LIN {X 0,Y 378.118,Z 312.233,A -85,B 0,C 180,E1 -14679.383,E2 -14679.383} C_VEL
LIN {X 0,Y 374.987,Z 310.362,A -85,B 0,C 180,E1 -14680.649,E2 -14680.649} C_VEL
LIN {X 0,Y 371.579,Z 307.37,A -85,B 0,C 180,E1 -14681.941,E2 -14681.941} C_VEL
LIN {X 0,Y 368.941,Z 304.589,A -85,B 0,C 180,E1 -14682.864,E2 -14682.864} C_VEL
LIN {X 0,Y 365.212,Z 301.597,A -85,B 0,C 180,E1 -14683.991,E2 -14683.991} C_VEL
LIN {X 0,Y 361.301,Z 297.475,A -85,B 0,C 180,E1 -14685.117,E2 -14685.117} C_VEL
LIN {X 0,Y 357.11,Z 293.614,A -85,B 0,C 180,E1 -14686.197,E2 -14686.197} C_VEL
LIN {X 0,Y 354.383,Z 290.674,A -85,B 0,C 180,E1 -14686.85,E2 -14686.85} C_VEL
LIN {X 0,Y 350.827,Z 287.024,A -85,B 0,C 180,E1 -14687.67,E2 -14687.67} C_VEL
LIN {X 0,Y 348.359,Z 284.254,A -85,B 0,C 180,E1 -14688.225,E2 -14688.225} C_VEL
LIN {X 0,Y 345.121,Z 280.43,A -85,B 0,C 180,E1 -14688.925,E2 -14688.925} C_VEL
LIN {X 0,Y 340.974,Z 275.499,A -85,B 0,C 180,E1 -14689.77,E2 -14689.77} C_VEL
LIN {X 0,Y 339.656,Z 273.734,A -85,B 0,C 180,E1 -14690.037,E2 -14690.037} C_VEL
LIN {X 0,Y 337.259,Z 270.621,A -85,B 0,C 180,E1 -14690.505,E2 -14690.505} C_VEL
LIN {X 0,Y 336.338,Z 269.13,A -85,B 0,C 180,E1 -14690.687,E2 -14690.687} C_VEL
LIN {X 0,Y 334.367,Z 266.713,A -85,B 0,C 180,E1 -14691.057,E2 -14691.057} C_VEL
LIN {X 0,Y 333.668,Z 264.421,A -85,B 0,C 180,E1 -14691.262,E2 -14691.262} C_VEL
LIN {X 0,Y 333.674,Z 264.419,A -85,B 0,C 180,E1 -14695.108,E2 -14695.108} C_VEL
LIN {X 0,Y 333.658,Z 264.421,A -85,B 0,C 180,E1 -14698.976,E2 -14698.976} C_VEL
LIN {X 0,Y 333.6,Z 264.429,A -85,B 0,C 180,E1 -14702.594,E2 -14702.594} C_VEL
LIN {X 0,Y 333.627,Z 264.428,A -85,B 0,C 180,E1 -14706.144,E2 -14706.144} C_VEL
LIN {X 0,Y 333.635,Z 264.424,A -85,B 0,C 180,E1 -14709.193,E2 -14709.193} C_VEL
LIN {X 0,Y 333.658,Z 264.42,A -85,B 0,C 180,E1 -14712.519,E2 -14712.519} C_VEL
LIN {X 0,Y 333.687,Z 264.419,A -85,B 0,C 180,E1 -14715.983,E2 -14715.983} C_VEL
LIN {X 0,Y 333.662,Z 264.423,A -85,B 0,C 180,E1 -14719.311,E2 -14719.311} C_VEL
LIN {X 0,Y 333.628,Z 264.427,A -85,B 0,C 180,E1 -14723.175,E2 -14723.175} C_VEL
LIN {X 0,Y 333.639,Z 264.428,A -85,B 0,C 180,E1 -14725.348,E2 -14725.348} C_VEL
LIN {X 0,Y 333.66,Z 264.422,A -85,B 0,C 180,E1 -14729.644,E2 -14729.644} C_VEL
LIN {X 0,Y 333.711,Z 264.414,A -85,B 0,C 180,E1 -14732.408,E2 -14732.408} C_VEL
LIN {X 0,Y 333.7,Z 264.419,A -85,B 0,C 180,E1 -14735.098,E2 -14735.098} C_VEL
LIN {X 0,Y 333.65,Z 264.425,A -85,B 0,C 180,E1 -14739.026,E2 -14739.026} C_VEL
LIN {X 0,Y 333.642,Z 264.421,A -85,B 0,C 180,E1 -14739.892,E2 -14739.892} C_VEL
LIN {X 0,Y 333.012,Z 264.505,A -85,B 0,C 180,E1 -14740.899,E2 -14740.899} C_VEL
LIN {X 0,Y 330.2,Z 264.856,A -85,B 0,C 180,E1 -14742.539,E2 -14742.539} C_VEL
LIN {X 0,Y 327.813,Z 265.154,A -85,B 0,C 180,E1 -14743.868,E2 -14743.868} C_VEL
LIN {X 0,Y 326.808,Z 265.277,A -85,B 0,C 180,E1 -14744.896,E2 -14744.896} C_VEL
LIN {X 0,Y 326.737,Z 265.283,A -85,B 0,C 180,E1 -14745.244,E2 -14745.244} C_VEL
LIN {X 0,Y 326.743,Z 265.284,A -85,B 0,C 180,E1 -14748.846,E2 -14748.846} C_VEL
LIN {X 0,Y 326.928,Z 265.264,A -85,B 0,C 180,E1 -14752.597,E2 -14752.597} C_VEL
LIN {X 0,Y 326.751,Z 265.28,A -85,B 0,C 180,E1 -14755.072,E2 -14755.072} C_VEL
LIN {X 0,Y 327.009,Z 265.244,A -85,B 0,C 180,E1 -14757.544,E2 -14757.544} C_VEL
LIN {X 0,Y 327.039,Z 265.244,A -85,B 0,C 180,E1 -14761.238,E2 -14761.238} C_VEL
LIN {X 0,Y 326.744,Z 265.283,A -85,B 0,C 180,E1 -14763.707,E2 -14763.707} C_VEL
LIN {X 0,Y 326.937,Z 265.263,A -85,B 0,C 180,E1 -14766.177,E2 -14766.177} C_VEL
LIN {X 0,Y 326.783,Z 265.281,A -85,B 0,C 180,E1 -14769.914,E2 -14769.914} C_VEL
LIN {X 0,Y 326.745,Z 265.285,A -85,B 0,C 180,E1 -14773.692,E2 -14773.692} C_VEL
LIN {X 0,Y 326.635,Z 265.299,A -85,B 0,C 180,E1 -14777.538,E2 -14777.538} C_VEL
LIN {X 0,Y 326.614,Z 265.301,A -85,B 0,C 180,E1 -14781.463,E2 -14781.463} C_VEL
LIN {X 0,Y 326.607,Z 265.304,A -85,B 0,C 180,E1 -14785.497,E2 -14785.497} C_VEL
LIN {X 0,Y 326.598,Z 265.301,A -85,B 0,C 180,E1 -14788.262,E2 -14788.262} C_VEL
LIN {X 0,Y 326.582,Z 265.306,A -85,B 0,C 180,E1 -14791.102,E2 -14791.102} C_VEL
LIN {X 0,Y 326.617,Z 265.301,A -85,B 0,C 180,E1 -14794.025,E2 -14794.025} C_VEL
LIN {X 0,Y 326.696,Z 265.699,A -85,B 0,C 180,E1 -14795.515,E2 -14795.515} C_VEL
LIN {X 0,Y 327.042,Z 268.418,A -85,B 0,C 180,E1 -14799.321,E2 -14799.321} C_VEL
LIN {X 0,Y 327.515,Z 271.566,A -85,B 0,C 180,E1 -14803.374,E2 -14803.374} C_VEL
LIN {X 0,Y 327.812,Z 274.541,A -85,B 0,C 180,E1 -14806.803,E2 -14806.803} C_VEL
LIN {X 0,Y 327.68,Z 277.535,A -85,B 0,C 180,E1 -14809.953,E2 -14809.953} C_VEL
LIN {X 0,Y 327.245,Z 280.671,A -85,B 0,C 180,E1 -14813.035,E2 -14813.035} C_VEL
LIN {X 0,Y 326.824,Z 283.847,A -85,B 0,C 180,E1 -14816.007,E2 -14816.007} C_VEL
LIN {X 0,Y 326.327,Z 287.744,A -85,B 0,C 180,E1 -14819.49,E2 -14819.49} C_VEL
LIN {X 0,Y 325.872,Z 291.916,A -85,B 0,C 180,E1 -14823.071,E2 -14823.071} C_VEL
LIN {X 0,Y 325.594,Z 295.184,A -85,B 0,C 180,E1 -14825.788,E2 -14825.788} C_VEL
LIN {X 0,Y 325.375,Z 297.414,A -85,B 0,C 180,E1 -14827.655,E2 -14827.655} C_VEL
LIN {X 0,Y 327.631,Z 306.627,A -85,B 0,C 180,E1 -14828.169,E2 -14828.169} C_VEL
LIN {X 0,Y 329.542,Z 316.235,A -85,B 0,C 180,E1 -14828.811,E2 -14828.811} C_VEL
LIN {X 0,Y 331.065,Z 325.863,A -85,B 0,C 180,E1 -14829.575,E2 -14829.575} C_VEL
LIN {X 0,Y 332.055,Z 334.461,A -85,B 0,C 180,E1 -14830.367,E2 -14830.367} C_VEL
LIN {X 0,Y 332.381,Z 339.384,A -85,B 0,C 180,E1 -14830.869,E2 -14830.869} C_VEL
LIN {X 0,Y 330.863,Z 351.576,A -85,B 0,C 180,E1 -14832.221,E2 -14832.221} C_VEL
LIN {X 0,Y 329.881,Z 359.328,A -85,B 0,C 180,E1 -14833.286,E2 -14833.286} C_VEL
LIN {X 0,Y 328.683,Z 368.467,A -85,B 0,C 180,E1 -14834.815,E2 -14834.815} C_VEL
LIN {X 0,Y 327.874,Z 374.673,A -85,B 0,C 180,E1 -14836.046,E2 -14836.046} C_VEL
LIN {X 0,Y 326.889,Z 381.211,A -85,B 0,C 180,E1 -14837.585,E2 -14837.585} C_VEL
LIN {X 0,Y 326.349,Z 385.716,A -85,B 0,C 180,E1 -14838.825,E2 -14838.825} C_VEL
LIN {X 0,Y 325.657,Z 391.211,A -85,B 0,C 180,E1 -14840.685,E2 -14840.685} C_VEL
LIN {X 0,Y 325.219,Z 395.539,A -85,B 0,C 180,E1 -14842.55,E2 -14842.55} C_VEL
LIN {X 0,Y 325.008,Z 398.409,A -85,B 0,C 180,E1 -14844.139,E2 -14844.139} C_VEL
LIN {X 0,Y 324.915,Z 401.1,A -85,B 0,C 180,E1 -14846.279,E2 -14846.279} C_VEL
LIN {X 0,Y 324.845,Z 402.158,A -85,B 0,C 180,E1 -14847.52,E2 -14847.52} C_VEL
LIN {X 0,Y 324.823,Z 402.747,A -85,B 0,C 180,E1 -14848.76,E2 -14848.76} C_VEL
LIN {X 0,Y 324.823,Z 402.747,A -85,B 0,C 180,E1 -14851.24,E2 -14851.24} C_VEL
LIN {X 0,Y 324.845,Z 402.158,A -85,B 0,C 180,E1 -14852.48,E2 -14852.48} C_VEL
LIN {X 0,Y 324.926,Z 399.709,A -85,B 0,C 180,E1 -14854.963,E2 -14854.963} C_VEL
LIN {X 0,Y 325.108,Z 396.757,A -85,B 0,C 180,E1 -14856.828,E2 -14856.828} C_VEL
LIN {X 0,Y 325.489,Z 392.766,A -85,B 0,C 180,E1 -14858.693,E2 -14858.693} C_VEL
LIN {X 0,Y 326.087,Z 387.633,A -85,B 0,C 180,E1 -14860.556,E2 -14860.556} C_VEL
LIN {X 0,Y 326.724,Z 382.367,A -85,B 0,C 180,E1 -14862.106,E2 -14862.106} C_VEL
LIN {X 0,Y 327.65,Z 376.049,A -85,B 0,C 180,E1 -14863.647,E2 -14863.647} C_VEL
LIN {X 0,Y 328.433,Z 370.094,A -85,B 0,C 180,E1 -14864.879,E2 -14864.879} C_VEL
LIN {X 0,Y 329.506,Z 362.015,A -85,B 0,C 180,E1 -14866.288,E2 -14866.288} C_VEL
LIN {X 0,Y 330.538,Z 353.845,A -85,B 0,C 180,E1 -14867.477,E2 -14867.477} C_VEL
LIN {X 0,Y 331.678,Z 345.117,A -85,B 0,C 180,E1 -14868.532,E2 -14868.532} C_VEL
LIN {X 0,Y 332.396,Z 337.747,A -85,B 0,C 180,E1 -14869.291,E2 -14869.291} C_VEL
LIN {X 0,Y 331.343,Z 327.774,A -85,B 0,C 180,E1 -14870.254,E2 -14870.254} C_VEL
LIN {X 0,Y 330.031,Z 319.039,A -85,B 0,C 180,E1 -14870.98,E2 -14870.98} C_VEL
LIN {X 0,Y 328.032,Z 308.528,A -85,B 0,C 180,E1 -14871.714,E2 -14871.714} C_VEL
LIN {X 0,Y 325.669,Z 299.128,A -85,B 0,C 180,E1 -14872.271,E2 -14872.271} C_VEL
LIN {X 0,Y 325.394,Z 297.387,A -85,B 0,C 180,E1 -14872.368,E2 -14872.368} C_VEL
LIN {X 0,Y 325.704,Z 293.555,A -85,B 0,C 180,E1 -14875.566,E2 -14875.566} C_VEL
LIN {X 0,Y 326.073,Z 290.285,A -85,B 0,C 180,E1 -14878.305,E2 -14878.305} C_VEL
LIN {X 0,Y 326.618,Z 285.433,A -85,B 0,C 180,E1 -14882.543,E2 -14882.543} C_VEL
LIN {X 0,Y 327.059,Z 282.248,A -85,B 0,C 180,E1 -14885.463,E2 -14885.463} C_VEL
LIN {X 0,Y 327.465,Z 279.094,A -85,B 0,C 180,E1 -14888.49,E2 -14888.49} C_VEL
LIN {X 0,Y 327.82,Z 275.972,A -85,B 0,C 180,E1 -14891.65,E2 -14891.65} C_VEL
LIN {X 0,Y 327.845,Z 274.426,A -85,B 0,C 180,E1 -14893.312,E2 -14893.312} C_VEL
LIN {X 0,Y 327.486,Z 271.384,A -85,B 0,C 180,E1 -14896.856,E2 -14896.856} C_VEL
LIN {X 0,Y 327.041,Z 268.391,A -85,B 0,C 180,E1 -14900.679,E2 -14900.679} C_VEL
LIN {X 0,Y 326.666,Z 265.471,A -85,B 0,C 180,E1 -14904.838,E2 -14904.838} C_VEL
LIN {X 0,Y 326.616,Z 265.3,A -85,B 0,C 180,E1 -14907.45,E2 -14907.45} C_VEL
LIN {X 0,Y 326.589,Z 265.305,A -85,B 0,C 180,E1 -14910.328,E2 -14910.328} C_VEL
LIN {X 0,Y 326.603,Z 265.301,A -85,B 0,C 180,E1 -14913.129,E2 -14913.129} C_VEL
LIN {X 0,Y 326.597,Z 265.301,A -85,B 0,C 180,E1 -14917.205,E2 -14917.205} C_VEL
LIN {X 0,Y 326.653,Z 265.293,A -85,B 0,C 180,E1 -14921.2,E2 -14921.2} C_VEL
LIN {X 0,Y 326.728,Z 265.284,A -85,B 0,C 180,E1 -14925.453,E2 -14925.453} C_VEL
LIN {X 0,Y 326.758,Z 265.28,A -85,B 0,C 180,E1 -14928.832,E2 -14928.832} C_VEL
LIN {X 0,Y 326.91,Z 265.261,A -85,B 0,C 180,E1 -14932.582,E2 -14932.582} C_VEL
LIN {X 0,Y 326.741,Z 265.282,A -85,B 0,C 180,E1 -14935.057,E2 -14935.057} C_VEL
LIN {X 0,Y 327.003,Z 265.253,A -85,B 0,C 180,E1 -14937.529,E2 -14937.529} C_VEL
LIN {X 0,Y 327.021,Z 265.245,A -85,B 0,C 180,E1 -14941.224,E2 -14941.224} C_VEL
LIN {X 0,Y 326.758,Z 265.282,A -85,B 0,C 180,E1 -14943.692,E2 -14943.692} C_VEL
LIN {X 0,Y 326.923,Z 265.259,A -85,B 0,C 180,E1 -14946.578,E2 -14946.578} C_VEL
LIN {X 0,Y 326.769,Z 265.279,A -85,B 0,C 180,E1 -14949.9,E2 -14949.9} C_VEL
LIN {X 0,Y 326.74,Z 265.283,A -85,B 0,C 180,E1 -14953.678,E2 -14953.678} C_VEL
LIN {X 0,Y 326.644,Z 265.296,A -85,B 0,C 180,E1 -14957.522,E2 -14957.522} C_VEL
LIN {X 0,Y 326.611,Z 265.297,A -85,B 0,C 180,E1 -14960.129,E2 -14960.129} C_VEL
LIN {X 0,Y 326.623,Z 265.296,A -85,B 0,C 180,E1 -14964.122,E2 -14964.122} C_VEL
LIN {X 0,Y 326.655,Z 265.297,A -85,B 0,C 180,E1 -14966.85,E2 -14966.85} C_VEL
LIN {X 0,Y 326.603,Z 265.303,A -85,B 0,C 180,E1 -14970.602,E2 -14970.602} C_VEL
LIN {X 0,Y 326.573,Z 265.303,A -85,B 0,C 180,E1 -14974.012,E2 -14974.012} C_VEL
LIN {X 0,Y 326.59,Z 265.301,A -85,B 0,C 180,E1 -14977.231,E2 -14977.231} C_VEL
LIN {X 0,Y 326.596,Z 265.303,A -85,B 0,C 180,E1 -14980.196,E2 -14980.196} C_VEL
LIN {X 0,Y 326.616,Z 265.298,A -85,B 0,C 180,E1 -14983.503,E2 -14983.503} C_VEL
LIN {X 0,Y 326.606,Z 265.299,A -85,B 0,C 180,E1 -14987.008,E2 -14987.008} C_VEL
LIN {X 0,Y 326.596,Z 265.301,A -85,B 0,C 180,E1 -14990.76,E2 -14990.76} C_VEL
LIN {X 0,Y 326.563,Z 265.306,A -85,B 0,C 180,E1 -14994.475,E2 -14994.475} C_VEL
LIN {X 0,Y 326.564,Z 265.306,A -85,B 0,C 180,E1 -14997.451,E2 -14997.451} C_VEL
LIN {X 0,Y 326.609,Z 265.301,A -85,B 0,C 180,E1 -15000.336,E2 -15000.336} C_VEL
LIN {X 0,Y 326.639,Z 265.296,A -85,B 0,C 180,E1 -15004.513,E2 -15004.513} C_VEL
LIN {X 0,Y 326.659,Z 265.306,A -85,B 0,C 180,E1 -15007.838,E2 -15007.838} C_VEL
LIN {X 0,Y 327.653,Z 268.102,A -85,B 0,C 180,E1 -15008.036,E2 -15008.036} C_VEL
LIN {X 0,Y 329.492,Z 270.637,A -85,B 0,C 180,E1 -15008.359,E2 -15008.359} C_VEL
LIN {X 0,Y 331.912,Z 274.086,A -85,B 0,C 180,E1 -15008.791,E2 -15008.791} C_VEL
LIN {X 0,Y 336.088,Z 279.409,A -85,B 0,C 180,E1 -15009.56,E2 -15009.56} C_VEL
LIN {X 0,Y 340.074,Z 284.308,A -85,B 0,C 180,E1 -15010.336,E2 -15010.336} C_VEL
LIN {X 0,Y 345.247,Z 290.242,A -85,B 0,C 180,E1 -15011.402,E2 -15011.402} C_VEL
LIN {X 0,Y 350.921,Z 296.303,A -85,B 0,C 180,E1 -15012.674,E2 -15012.674} C_VEL
LIN {X 0,Y 353.867,Z 299.363,A -85,B 0,C 180,E1 -15013.385,E2 -15013.385} C_VEL
LIN {X 0,Y 358.117,Z 303.441,A -85,B 0,C 180,E1 -15014.474,E2 -15014.474} C_VEL
LIN {X 0,Y 360.414,Z 305.696,A -85,B 0,C 180,E1 -15015.099,E2 -15015.099} C_VEL
LIN {X 0,Y 364.679,Z 309.798,A -85,B 0,C 180,E1 -15016.367,E2 -15016.367} C_VEL
LIN {X 0,Y 367.684,Z 312.27,A -85,B 0,C 180,E1 -15017.333,E2 -15017.333} C_VEL
LIN {X 0,Y 370.703,Z 315.447,A -85,B 0,C 180,E1 -15018.461,E2 -15018.461} C_VEL
LIN {X 0,Y 372.499,Z 316.817,A -85,B 0,C 180,E1 -15019.125,E2 -15019.125} C_VEL
LIN {X 0,Y 375.47,Z 318.694,A -85,B 0,C 180,E1 -15020.302,E2 -15020.302} C_VEL
LIN {X 0,Y 378.606,Z 322.035,A -85,B 0,C 180,E1 -15021.956,E2 -15021.956} C_VEL
LIN {X 0,Y 381.325,Z 324.417,A -85,B 0,C 180,E1 -15023.651,E2 -15023.651} C_VEL
LIN {X 0,Y 382.838,Z 325.369,A -85,B 0,C 180,E1 -15024.734,E2 -15024.734} C_VEL
LIN {X 0,Y 384.098,Z 325.94,A -85,B 0,C 180,E1 -15025.803,E2 -15025.803} C_VEL
LIN {X 0,Y 385.138,Z 326.178,A -85,B 0,C 180,E1 -15026.862,E2 -15026.862} C_VEL
LIN {X 0,Y 385.873,Z 326.376,A -85,B 0,C 180,E1 -15027.912,E2 -15027.912} C_VEL
LIN {X 0,Y 386.479,Z 326.455,A -85,B 0,C 180,E1 -15029.734,E2 -15029.734} C_VEL
LIN {X 0,Y 386.344,Z 326.417,A -85,B 0,C 180,E1 -15031.042,E2 -15031.042} C_VEL
LIN {X 0,Y 385.873,Z 326.359,A -85,B 0,C 180,E1 -15032.088,E2 -15032.088} C_VEL
LIN {X 0,Y 385.147,Z 326.153,A -85,B 0,C 180,E1 -15033.138,E2 -15033.138} C_VEL
LIN {X 0,Y 384.113,Z 325.938,A -85,B 0,C 180,E1 -15034.197,E2 -15034.197} C_VEL
LIN {X 0,Y 381.631,Z 324.642,A -85,B 0,C 180,E1 -15036.132,E2 -15036.132} C_VEL
LIN {X 0,Y 379.595,Z 323.032,A -85,B 0,C 180,E1 -15037.446,E2 -15037.446} C_VEL
LIN {X 0,Y 377,Z 320.236,A -85,B 0,C 180,E1 -15038.94,E2 -15038.94} C_VEL
LIN {X 0,Y 375.398,Z 318.661,A -85,B 0,C 180,E1 -15039.7,E2 -15039.7} C_VEL
LIN {X 0,Y 372.189,Z 316.659,A -85,B 0,C 180,E1 -15040.966,E2 -15040.966} C_VEL
LIN {X 0,Y 368.327,Z 313.092,A -85,B 0,C 180,E1 -15042.418,E2 -15042.418} C_VEL
LIN {X 0,Y 366.165,Z 310.906,A -85,B 0,C 180,E1 -15043.166,E2 -15043.166} C_VEL
LIN {X 0,Y 362.128,Z 307.55,A -85,B 0,C 180,E1 -15044.384,E2 -15044.384} C_VEL
LIN {X 0,Y 358.612,Z 303.811,A -85,B 0,C 180,E1 -15045.398,E2 -15045.398} C_VEL
LIN {X 0,Y 354.435,Z 300.023,A -85,B 0,C 180,E1 -15046.464,E2 -15046.464} C_VEL
LIN {X 0,Y 351.099,Z 296.469,A -85,B 0,C 180,E1 -15047.283,E2 -15047.283} C_VEL
LIN {X 0,Y 347.136,Z 292.244,A -85,B 0,C 180,E1 -15048.194,E2 -15048.194} C_VEL
LIN {X 0,Y 341.992,Z 286.589,A -85,B 0,C 180,E1 -15049.275,E2 -15049.275} C_VEL
LIN {X 0,Y 337.043,Z 280.652,A -85,B 0,C 180,E1 -15050.256,E2 -15050.256} C_VEL
LIN {X 0,Y 333.214,Z 275.765,A -85,B 0,C 180,E1 -15050.979,E2 -15050.979} C_VEL
LIN {X 0,Y 329.744,Z 271.114,A -85,B 0,C 180,E1 -15051.591,E2 -15051.591} C_VEL
LIN {X 0,Y 328.709,Z 269.48,A -85,B 0,C 180,E1 -15051.782,E2 -15051.782} C_VEL
LIN {X 0,Y 327.076,Z 266.985,A -85,B 0,C 180,E1 -15052.066,E2 -15052.066} C_VEL
LIN {X 0,Y 326.659,Z 265.297,A -85,B 0,C 180,E1 -15052.193,E2 -15052.193} C_VEL
LIN {X 0,Y 326.639,Z 265.296,A -85,B 0,C 180,E1 -15055.487,E2 -15055.487} C_VEL
LIN {X 0,Y 326.609,Z 265.301,A -85,B 0,C 180,E1 -15059.664,E2 -15059.664} C_VEL
LIN {X 0,Y 326.572,Z 265.303,A -85,B 0,C 180,E1 -15062.952,E2 -15062.952} C_VEL
LIN {X 0,Y 326.582,Z 265.302,A -85,B 0,C 180,E1 -15067.052,E2 -15067.052} C_VEL
LIN {X 0,Y 326.589,Z 265.303,A -85,B 0,C 180,E1 -15070.208,E2 -15070.208} C_VEL
LIN {X 0,Y 326.614,Z 265.301,A -85,B 0,C 180,E1 -15073.516,E2 -15073.516} C_VEL
LIN {X 0,Y 326.609,Z 265.299,A -85,B 0,C 180,E1 -15077.021,E2 -15077.021} C_VEL
LIN {X 0,Y 326.604,Z 265.3,A -85,B 0,C 180,E1 -15080.773,E2 -15080.773} C_VEL
LIN {X 0,Y 326.576,Z 265.302,A -85,B 0,C 180,E1 -15084.487,E2 -15084.487} C_VEL
LIN {X 0,Y 326.575,Z 265.306,A -85,B 0,C 180,E1 -15087.463,E2 -15087.463} C_VEL
LIN {X 0,Y 326.618,Z 265.297,A -85,B 0,C 180,E1 -15090.347,E2 -15090.347} C_VEL
LIN {X 0,Y 326.664,Z 265.292,A -85,B 0,C 180,E1 -15094.524,E2 -15094.524} C_VEL
LIN {X 0,Y 326.596,Z 265.302,A -85,B 0,C 180,E1 -15098.551,E2 -15098.551} C_VEL
LIN {X 0,Y 326.687,Z 265.291,A -85,B 0,C 180,E1 -15101.183,E2 -15101.183} C_VEL
LIN {X 0,Y 326.737,Z 265.283,A -85,B 0,C 180,E1 -15105.244,E2 -15105.244} C_VEL
LIN {X 0,Y 326.09,Z 265.366,A -85,B 0,C 180,E1 -15106.273,E2 -15106.273} C_VEL
LIN {X 0,Y 323.219,Z 265.721,A -85,B 0,C 180,E1 -15107.947,E2 -15107.947} C_VEL
LIN {X 0,Y 320.804,Z 266.021,A -85,B 0,C 180,E1 -15109.304,E2 -15109.304} C_VEL
LIN {X 0,Y 319.814,Z 266.147,A -85,B 0,C 180,E1 -15110.355,E2 -15110.355} C_VEL
LIN {X 0,Y 319.76,Z 266.149,A -85,B 0,C 180,E1 -15110.711,E2 -15110.711} C_VEL
LIN {X 0,Y 319.904,Z 266.134,A -85,B 0,C 180,E1 -15113.701,E2 -15113.701} C_VEL
LIN {X 0,Y 319.955,Z 266.121,A -85,B 0,C 180,E1 -15117.49,E2 -15117.49} C_VEL
LIN {X 0,Y 320.007,Z 266.12,A -85,B 0,C 180,E1 -15121.266,E2 -15121.266} C_VEL
LIN {X 0,Y 319.711,Z 266.158,A -85,B 0,C 180,E1 -15125.052,E2 -15125.052} C_VEL
LIN {X 0,Y 319.85,Z 266.142,A -85,B 0,C 180,E1 -15127.583,E2 -15127.583} C_VEL
LIN {X 0,Y 319.714,Z 266.159,A -85,B 0,C 180,E1 -15131.417,E2 -15131.417} C_VEL
LIN {X 0,Y 319.667,Z 266.164,A -85,B 0,C 180,E1 -15134.684,E2 -15134.684} C_VEL
LIN {X 0,Y 319.591,Z 266.177,A -85,B 0,C 180,E1 -15137.937,E2 -15137.937} C_VEL
LIN {X 0,Y 319.569,Z 266.179,A -85,B 0,C 180,E1 -15141.961,E2 -15141.961} C_VEL
LIN {X 0,Y 319.557,Z 266.179,A -85,B 0,C 180,E1 -15146.101,E2 -15146.101} C_VEL
LIN {X 0,Y 319.533,Z 266.183,A -85,B 0,C 180,E1 -15148.946,E2 -15148.946} C_VEL
LIN {X 0,Y 319.533,Z 266.185,A -85,B 0,C 180,E1 -15151.868,E2 -15151.868} C_VEL
LIN {X 0,Y 319.639,Z 266.435,A -85,B 0,C 180,E1 -15154.873,E2 -15154.873} C_VEL
LIN {X 0,Y 319.891,Z 268.555,A -85,B 0,C 180,E1 -15157.97,E2 -15157.97} C_VEL
LIN {X 0,Y 320.3,Z 271.316,A -85,B 0,C 180,E1 -15161.754,E2 -15161.754} C_VEL
LIN {X 0,Y 320.673,Z 274.349,A -85,B 0,C 180,E1 -15165.468,E2 -15165.468} C_VEL
LIN {X 0,Y 320.773,Z 276.743,A -85,B 0,C 180,E1 -15168.16,E2 -15168.16} C_VEL
LIN {X 0,Y 320.571,Z 278.992,A -85,B 0,C 180,E1 -15170.523,E2 -15170.523} C_VEL
LIN {X 0,Y 319.987,Z 282.879,A -85,B 0,C 180,E1 -15174.363,E2 -15174.363} C_VEL
LIN {X 0,Y 319.422,Z 286.912,A -85,B 0,C 180,E1 -15178.127,E2 -15178.127} C_VEL
LIN {X 0,Y 318.984,Z 291.03,A -85,B 0,C 180,E1 -15181.808,E2 -15181.808} C_VEL
LIN {X 0,Y 318.557,Z 294.987,A -85,B 0,C 180,E1 -15185.218,E2 -15185.218} C_VEL
LIN {X 0,Y 318.335,Z 297.213,A -85,B 0,C 180,E1 -15187.127,E2 -15187.127} C_VEL
LIN {X 0,Y 320.755,Z 307.18,A -85,B 0,C 180,E1 -15187.714,E2 -15187.714} C_VEL
LIN {X 0,Y 322.582,Z 315.881,A -85,B 0,C 180,E1 -15188.322,E2 -15188.322} C_VEL
LIN {X 0,Y 324.268,Z 326.481,A -85,B 0,C 180,E1 -15189.196,E2 -15189.196} C_VEL
LIN {X 0,Y 325.264,Z 335.884,A -85,B 0,C 180,E1 -15190.105,E2 -15190.105} C_VEL
LIN {X 0,Y 325.512,Z 340.784,A -85,B 0,C 180,E1 -15190.613,E2 -15190.613} C_VEL
LIN {X 0,Y 324.085,Z 351.364,A -85,B 0,C 180,E1 -15191.837,E2 -15191.837} C_VEL
LIN {X 0,Y 323.002,Z 359.496,A -85,B 0,C 180,E1 -15192.984,E2 -15192.984} C_VEL
LIN {X 0,Y 322.054,Z 366.823,A -85,B 0,C 180,E1 -15194.209,E2 -15194.209} C_VEL
LIN {X 0,Y 320.974,Z 374.461,A -85,B 0,C 180,E1 -15195.74,E2 -15195.74} C_VEL
LIN {X 0,Y 319.933,Z 380.999,A -85,B 0,C 180,E1 -15197.311,E2 -15197.311} C_VEL
LIN {X 0,Y 319.33,Z 385.503,A -85,B 0,C 180,E1 -15198.576,E2 -15198.576} C_VEL
LIN {X 0,Y 318.637,Z 390.999,A -85,B 0,C 180,E1 -15200.478,E2 -15200.478} C_VEL
LIN {X 0,Y 318.142,Z 395.327,A -85,B 0,C 180,E1 -15202.383,E2 -15202.383} C_VEL
LIN {X 0,Y 317.896,Z 398.501,A -85,B 0,C 180,E1 -15204.222,E2 -15204.222} C_VEL
LIN {X 0,Y 317.824,Z 400.888,A -85,B 0,C 180,E1 -15206.196,E2 -15206.196} C_VEL
LIN {X 0,Y 317.768,Z 401.947,A -85,B 0,C 180,E1 -15207.465,E2 -15207.465} C_VEL
LIN {X 0,Y 317.736,Z 402.536,A -85,B 0,C 180,E1 -15208.733,E2 -15208.733} C_VEL
LIN {X 0,Y 317.736,Z 402.536,A -85,B 0,C 180,E1 -15211.267,E2 -15211.267} C_VEL
LIN {X 0,Y 317.768,Z 401.947,A -85,B 0,C 180,E1 -15212.535,E2 -15212.535} C_VEL
LIN {X 0,Y 317.844,Z 399.498,A -85,B 0,C 180,E1 -15215.074,E2 -15215.074} C_VEL
LIN {X 0,Y 318.035,Z 396.545,A -85,B 0,C 180,E1 -15216.981,E2 -15216.981} C_VEL
LIN {X 0,Y 318.44,Z 392.554,A -85,B 0,C 180,E1 -15218.887,E2 -15218.887} C_VEL
LIN {X 0,Y 319.072,Z 387.421,A -85,B 0,C 180,E1 -15220.791,E2 -15220.791} C_VEL
LIN {X 0,Y 319.762,Z 382.155,A -85,B 0,C 180,E1 -15222.374,E2 -15222.374} C_VEL
LIN {X 0,Y 320.739,Z 375.837,A -85,B 0,C 180,E1 -15223.947,E2 -15223.947} C_VEL
LIN {X 0,Y 321.548,Z 369.882,A -85,B 0,C 180,E1 -15225.205,E2 -15225.205} C_VEL
LIN {X 0,Y 322.568,Z 362.564,A -85,B 0,C 180,E1 -15226.519,E2 -15226.519} C_VEL
LIN {X 0,Y 323.602,Z 354.768,A -85,B 0,C 180,E1 -15227.701,E2 -15227.701} C_VEL
LIN {X 0,Y 324.749,Z 346.256,A -85,B 0,C 180,E1 -15228.778,E2 -15228.778} C_VEL
LIN {X 0,Y 325.585,Z 339.17,A -85,B 0,C 180,E1 -15229.547,E2 -15229.547} C_VEL
LIN {X 0,Y 324.513,Z 328.622,A -85,B 0,C 180,E1 -15230.613,E2 -15230.613} C_VEL
LIN {X 0,Y 322.95,Z 318.107,A -85,B 0,C 180,E1 -15231.508,E2 -15231.508} C_VEL
LIN {X 0,Y 320.929,Z 307.94,A -85,B 0,C 180,E1 -15232.237,E2 -15232.237} C_VEL
LIN {X 0,Y 318.336,Z 297.213,A -85,B 0,C 180,E1 -15232.873,E2 -15232.873} C_VEL
LIN {X 0,Y 318.672,Z 293.356,A -85,B 0,C 180,E1 -15236.172,E2 -15236.172} C_VEL
LIN {X 0,Y 319.05,Z 290.114,A -85,B 0,C 180,E1 -15238.987,E2 -15238.987} C_VEL
LIN {X 0,Y 319.422,Z 286.9,A -85,B 0,C 180,E1 -15241.873,E2 -15241.873} C_VEL
LIN {X 0,Y 320.014,Z 282.866,A -85,B 0,C 180,E1 -15245.644,E2 -15245.644} C_VEL
LIN {X 0,Y 320.572,Z 278.991,A -85,B 0,C 180,E1 -15249.477,E2 -15249.477} C_VEL
LIN {X 0,Y 320.793,Z 275.883,A -85,B 0,C 180,E1 -15252.777,E2 -15252.777} C_VEL
LIN {X 0,Y 320.513,Z 272.817,A -85,B 0,C 180,E1 -15256.352,E2 -15256.352} C_VEL
LIN {X 0,Y 320.09,Z 269.859,A -85,B 0,C 180,E1 -15260.215,E2 -15260.215} C_VEL
LIN {X 0,Y 319.687,Z 266.875,A -85,B 0,C 180,E1 -15264.429,E2 -15264.429} C_VEL
LIN {X 0,Y 319.639,Z 266.424,A -85,B 0,C 180,E1 -15265.127,E2 -15265.127} C_VEL
LIN {X 0,Y 319.533,Z 266.184,A -85,B 0,C 180,E1 -15268.132,E2 -15268.132} C_VEL
LIN {X 0,Y 319.553,Z 266.179,A -85,B 0,C 180,E1 -15271.608,E2 -15271.608} C_VEL
LIN {X 0,Y 319.532,Z 266.182,A -85,B 0,C 180,E1 -15275.292,E2 -15275.292} C_VEL
LIN {X 0,Y 319.569,Z 266.18,A -85,B 0,C 180,E1 -15278.039,E2 -15278.039} C_VEL
LIN {X 0,Y 319.591,Z 266.177,A -85,B 0,C 180,E1 -15282.063,E2 -15282.063} C_VEL
LIN {X 0,Y 319.712,Z 266.162,A -85,B 0,C 180,E1 -15286,E2 -15286} C_VEL
LIN {X 0,Y 319.735,Z 266.159,A -85,B 0,C 180,E1 -15289.865,E2 -15289.865} C_VEL
LIN {X 0,Y 319.894,Z 266.139,A -85,B 0,C 180,E1 -15293.686,E2 -15293.686} C_VEL
LIN {X 0,Y 319.949,Z 266.131,A -85,B 0,C 180,E1 -15297.475,E2 -15297.475} C_VEL
LIN {X 0,Y 319.991,Z 266.121,A -85,B 0,C 180,E1 -15301.251,E2 -15301.251} C_VEL
LIN {X 0,Y 319.708,Z 266.16,A -85,B 0,C 180,E1 -15303.774,E2 -15303.774} C_VEL
LIN {X 0,Y 319.886,Z 266.135,A -85,B 0,C 180,E1 -15306.566,E2 -15306.566} C_VEL
LIN {X 0,Y 319.721,Z 266.156,A -85,B 0,C 180,E1 -15310.12,E2 -15310.12} C_VEL
LIN {X 0,Y 319.714,Z 266.157,A -85,B 0,C 180,E1 -15313.985,E2 -15313.985} C_VEL
LIN {X 0,Y 319.604,Z 266.171,A -85,B 0,C 180,E1 -15317.921,E2 -15317.921} C_VEL
LIN {X 0,Y 319.545,Z 266.178,A -85,B 0,C 180,E1 -15321.947,E2 -15321.947} C_VEL
LIN {X 0,Y 319.591,Z 266.172,A -85,B 0,C 180,E1 -15326.082,E2 -15326.082} C_VEL
LIN {X 0,Y 319.551,Z 266.182,A -85,B 0,C 180,E1 -15328.927,E2 -15328.927} C_VEL
LIN {X 0,Y 319.498,Z 266.184,A -85,B 0,C 180,E1 -15331.855,E2 -15331.855} C_VEL
LIN {X 0,Y 319.544,Z 266.178,A -85,B 0,C 180,E1 -15335.535,E2 -15335.535} C_VEL
LIN {X 0,Y 319.544,Z 266.18,A -85,B 0,C 180,E1 -15338,E2 -15338} C_VEL
LIN {X 0,Y 319.561,Z 266.177,A -85,B 0,C 180,E1 -15341.605,E2 -15341.605} C_VEL
LIN {X 0,Y 319.603,Z 266.171,A -85,B 0,C 180,E1 -15345.279,E2 -15345.279} C_VEL
LIN {X 0,Y 319.538,Z 266.181,A -85,B 0,C 180,E1 -15348.714,E2 -15348.714} C_VEL
LIN {X 0,Y 319.534,Z 266.184,A -85,B 0,C 180,E1 -15352.338,E2 -15352.338} C_VEL
LIN {X 0,Y 319.51,Z 266.183,A -85,B 0,C 180,E1 -15355.118,E2 -15355.118} C_VEL
LIN {X 0,Y 319.522,Z 266.182,A -85,B 0,C 180,E1 -15359.052,E2 -15359.052} C_VEL
LIN {X 0,Y 319.555,Z 266.179,A -85,B 0,C 180,E1 -15362.494,E2 -15362.494} C_VEL
LIN {X 0,Y 319.574,Z 266.178,A -85,B 0,C 180,E1 -15365.302,E2 -15365.302} C_VEL
LIN {X 0,Y 319.61,Z 266.173,A -85,B 0,C 180,E1 -15367.027,E2 -15367.027} C_VEL
LIN {X 0,Y 320.674,Z 269.144,A -85,B 0,C 180,E1 -15367.226,E2 -15367.226} C_VEL
LIN {X 0,Y 322.157,Z 271.338,A -85,B 0,C 180,E1 -15367.45,E2 -15367.45} C_VEL
LIN {X 0,Y 324.428,Z 274.689,A -85,B 0,C 180,E1 -15367.817,E2 -15367.817} C_VEL
LIN {X 0,Y 327.539,Z 279.052,A -85,B 0,C 180,E1 -15368.327,E2 -15368.327} C_VEL
LIN {X 0,Y 332.288,Z 284.974,A -85,B 0,C 180,E1 -15369.174,E2 -15369.174} C_VEL
LIN {X 0,Y 336.349,Z 289.91,A -85,B 0,C 180,E1 -15369.955,E2 -15369.955} C_VEL
LIN {X 0,Y 341.731,Z 296.056,A -85,B 0,C 180,E1 -15371.059,E2 -15371.059} C_VEL
LIN {X 0,Y 347.373,Z 302.107,A -85,B 0,C 180,E1 -15372.334,E2 -15372.334} C_VEL
LIN {X 0,Y 350.5,Z 305.354,A -85,B 0,C 180,E1 -15373.09,E2 -15373.09} C_VEL
LIN {X 0,Y 355.015,Z 309.675,A -85,B 0,C 180,E1 -15374.252,E2 -15374.252} C_VEL
LIN {X 0,Y 360.386,Z 315.045,A -85,B 0,C 180,E1 -15375.805,E2 -15375.805} C_VEL
LIN {X 0,Y 364.886,Z 318.868,A -85,B 0,C 180,E1 -15377.223,E2 -15377.223} C_VEL
LIN {X 0,Y 367.679,Z 321.741,A -85,B 0,C 180,E1 -15378.273,E2 -15378.273} C_VEL
LIN {X 0,Y 371.402,Z 324.359,A -85,B 0,C 180,E1 -15379.679,E2 -15379.679} C_VEL
LIN {X 0,Y 373.699,Z 326.209,A -85,B 0,C 180,E1 -15380.696,E2 -15380.696} C_VEL
LIN {X 0,Y 376.827,Z 329.568,A -85,B 0,C 180,E1 -15382.499,E2 -15382.499} C_VEL
LIN {X 0,Y 378.571,Z 330.947,A -85,B 0,C 180,E1 -15383.605,E2 -15383.605} C_VEL
LIN {X 0,Y 380.766,Z 332.224,A -85,B 0,C 180,E1 -15385.23,E2 -15385.23} C_VEL
LIN {X 0,Y 382.485,Z 332.74,A -85,B 0,C 180,E1 -15386.84,E2 -15386.84} C_VEL
LIN {X 0,Y 383.244,Z 332.949,A -85,B 0,C 180,E1 -15387.898,E2 -15387.898} C_VEL
LIN {X 0,Y 383.734,Z 333.009,A -85,B 0,C 180,E1 -15388.951,E2 -15388.951} C_VEL
LIN {X 0,Y 383.886,Z 333.049,A -85,B 0,C 180,E1 -15390,E2 -15390} C_VEL
LIN {X 0,Y 383.725,Z 333.003,A -85,B 0,C 180,E1 -15391.049,E2 -15391.049} C_VEL
LIN {X 0,Y 383.235,Z 332.95,A -85,B 0,C 180,E1 -15392.102,E2 -15392.102} C_VEL
LIN {X 0,Y 382.491,Z 332.724,A -85,B 0,C 180,E1 -15393.16,E2 -15393.16} C_VEL
LIN {X 0,Y 380.768,Z 332.205,A -85,B 0,C 180,E1 -15394.774,E2 -15394.774} C_VEL
LIN {X 0,Y 378.558,Z 330.954,A -85,B 0,C 180,E1 -15396.395,E2 -15396.395} C_VEL
LIN {X 0,Y 376.064,Z 328.756,A -85,B 0,C 180,E1 -15397.983,E2 -15397.983} C_VEL
LIN {X 0,Y 372.696,Z 325.246,A -85,B 0,C 180,E1 -15399.771,E2 -15399.771} C_VEL
LIN {X 0,Y 369.713,Z 323.369,A -85,B 0,C 180,E1 -15400.958,E2 -15400.958} C_VEL
LIN {X 0,Y 366.503,Z 320.578,A -85,B 0,C 180,E1 -15402.177,E2 -15402.177} C_VEL
LIN {X 0,Y 361.742,Z 316.162,A -85,B 0,C 180,E1 -15403.775,E2 -15403.775} C_VEL
LIN {X 0,Y 358.439,Z 313.187,A -85,B 0,C 180,E1 -15404.767,E2 -15404.767} C_VEL
LIN {X 0,Y 355.431,Z 310.006,A -85,B 0,C 180,E1 -15405.642,E2 -15405.642} C_VEL
LIN {X 0,Y 350.626,Z 305.484,A -85,B 0,C 180,E1 -15406.88,E2 -15406.88} C_VEL
LIN {X 0,Y 347.035,Z 301.806,A -85,B 0,C 180,E1 -15407.747,E2 -15407.747} C_VEL
LIN {X 0,Y 340.82,Z 295.137,A -85,B 0,C 180,E1 -15409.124,E2 -15409.124} C_VEL
LIN {X 0,Y 333.372,Z 286.437,A -85,B 0,C 180,E1 -15410.619,E2 -15410.619} C_VEL
LIN {X 0,Y 328.823,Z 280.611,A -85,B 0,C 180,E1 -15411.453,E2 -15411.453} C_VEL
LIN {X 0,Y 325.211,Z 275.892,A -85,B 0,C 180,E1 -15412.062,E2 -15412.062} C_VEL
LIN {X 0,Y 322.15,Z 271.367,A -85,B 0,C 180,E1 -15412.55,E2 -15412.55} C_VEL
LIN {X 0,Y 319.945,Z 267.598,A -85,B 0,C 180,E1 -15412.889,E2 -15412.889} C_VEL
LIN {X 0,Y 319.592,Z 266.175,A -85,B 0,C 180,E1 -15412.972,E2 -15412.972} C_VEL
LIN {X 0,Y 319.582,Z 266.179,A -85,B 0,C 180,E1 -15416.092,E2 -15416.092} C_VEL
LIN {X 0,Y 319.537,Z 266.18,A -85,B 0,C 180,E1 -15418.938,E2 -15418.938} C_VEL
LIN {X 0,Y 319.487,Z 266.19,A -85,B 0,C 180,E1 -15421.866,E2 -15421.866} C_VEL
LIN {X 0,Y 319.53,Z 266.183,A -85,B 0,C 180,E1 -15425.548,E2 -15425.548} C_VEL
LIN {X 0,Y 319.535,Z 266.184,A -85,B 0,C 180,E1 -15428.013,E2 -15428.013} C_VEL
LIN {X 0,Y 319.557,Z 266.181,A -85,B 0,C 180,E1 -15431.618,E2 -15431.618} C_VEL
LIN {X 0,Y 319.603,Z 266.173,A -85,B 0,C 180,E1 -15435.291,E2 -15435.291} C_VEL
LIN {X 0,Y 319.543,Z 266.179,A -85,B 0,C 180,E1 -15438.727,E2 -15438.727} C_VEL
LIN {X 0,Y 319.544,Z 266.179,A -85,B 0,C 180,E1 -15442.351,E2 -15442.351} C_VEL
LIN {X 0,Y 319.525,Z 266.184,A -85,B 0,C 180,E1 -15445.13,E2 -15445.13} C_VEL
LIN {X 0,Y 319.535,Z 266.184,A -85,B 0,C 180,E1 -15449.067,E2 -15449.067} C_VEL
LIN {X 0,Y 319.577,Z 266.175,A -85,B 0,C 180,E1 -15452.505,E2 -15452.505} C_VEL
LIN {X 0,Y 319.578,Z 266.177,A -85,B 0,C 180,E1 -15455.311,E2 -15455.311} C_VEL
LIN {X 0,Y 319.565,Z 266.175,A -85,B 0,C 180,E1 -15459.407,E2 -15459.407} C_VEL
LIN {X 0,Y 319.604,Z 266.171,A -85,B 0,C 180,E1 -15462.079,E2 -15462.079} C_VEL
LIN {X 0,Y 319.714,Z 266.157,A -85,B 0,C 180,E1 -15466.015,E2 -15466.015} C_VEL
LIN {X 0,Y 319.721,Z 266.156,A -85,B 0,C 180,E1 -15469.88,E2 -15469.88} C_VEL
LIN {X 0,Y 319.76,Z 266.149,A -85,B 0,C 180,E1 -15470.711,E2 -15470.711} C_VEL
LIN {X 0,Y 319.482,Z 266.187,A -85,B 0,C 180,E1 -15471.414,E2 -15471.414} C_VEL
LIN {X 0,Y 317.51,Z 266.44,A -85,B 0,C 180,E1 -15472.793,E2 -15472.793} C_VEL
LIN {X 0,Y 313.709,Z 266.915,A -85,B 0,C 180,E1 -15474.858,E2 -15474.858} C_VEL
LIN {X 0,Y 312.719,Z 267.031,A -85,B 0,C 180,E1 -15475.933,E2 -15475.933} C_VEL
LIN {X 0,Y 312.68,Z 267.032,A -85,B 0,C 180,E1 -15476.298,E2 -15476.298} C_VEL
LIN {X 0,Y 312.96,Z 266.996,A -85,B 0,C 180,E1 -15478.721,E2 -15478.721} C_VEL
LIN {X 0,Y 312.974,Z 266.996,A -85,B 0,C 180,E1 -15481.294,E2 -15481.294} C_VEL
LIN {X 0,Y 312.836,Z 267.017,A -85,B 0,C 180,E1 -15486.457,E2 -15486.457} C_VEL
LIN {X 0,Y 312.751,Z 267.025,A -85,B 0,C 180,E1 -15489.057,E2 -15489.057} C_VEL
LIN {X 0,Y 312.626,Z 267.041,A -85,B 0,C 180,E1 -15492.998,E2 -15492.998} C_VEL
LIN {X 0,Y 312.574,Z 267.051,A -85,B 0,C 180,E1 -15495.66,E2 -15495.66} C_VEL
LIN {X 0,Y 312.534,Z 267.057,A -85,B 0,C 180,E1 -15499.72,E2 -15499.72} C_VEL
LIN {X 0,Y 312.521,Z 267.054,A -85,B 0,C 180,E1 -15502.78,E2 -15502.78} C_VEL
LIN {X 0,Y 312.49,Z 267.058,A -85,B 0,C 180,E1 -15506.738,E2 -15506.738} C_VEL
LIN {X 0,Y 312.478,Z 267.065,A -85,B 0,C 180,E1 -15509.664,E2 -15509.664} C_VEL
LIN {X 0,Y 312.541,Z 267.055,A -85,B 0,C 180,E1 -15513.696,E2 -15513.696} C_VEL
LIN {X 0,Y 312.707,Z 268.308,A -85,B 0,C 180,E1 -15515.994,E2 -15515.994} C_VEL
LIN {X 0,Y 313.105,Z 271.25,A -85,B 0,C 180,E1 -15520.257,E2 -15520.257} C_VEL
LIN {X 0,Y 313.514,Z 274.156,A -85,B 0,C 180,E1 -15524.028,E2 -15524.028} C_VEL
LIN {X 0,Y 313.746,Z 277.243,A -85,B 0,C 180,E1 -15527.671,E2 -15527.671} C_VEL
LIN {X 0,Y 313.42,Z 280.444,A -85,B 0,C 180,E1 -15531.108,E2 -15531.108} C_VEL
LIN {X 0,Y 312.961,Z 283.587,A -85,B 0,C 180,E1 -15534.278,E2 -15534.278} C_VEL
LIN {X 0,Y 312.452,Z 286.77,A -85,B 0,C 180,E1 -15537.328,E2 -15537.328} C_VEL
LIN {X 0,Y 312.064,Z 289.971,A -85,B 0,C 180,E1 -15540.3,E2 -15540.3} C_VEL
LIN {X 0,Y 311.669,Z 293.193,A -85,B 0,C 180,E1 -15543.193,E2 -15543.193} C_VEL
LIN {X 0,Y 311.325,Z 297.107,A -85,B 0,C 180,E1 -15546.593,E2 -15546.593} C_VEL
LIN {X 0,Y 313.531,Z 306.067,A -85,B 0,C 180,E1 -15547.128,E2 -15547.128} C_VEL
LIN {X 0,Y 315.454,Z 314.721,A -85,B 0,C 180,E1 -15547.745,E2 -15547.745} C_VEL
LIN {X 0,Y 317.095,Z 324.833,A -85,B 0,C 180,E1 -15548.583,E2 -15548.583} C_VEL
LIN {X 0,Y 318.2,Z 334.022,A -85,B 0,C 180,E1 -15549.475,E2 -15549.475} C_VEL
LIN {X 0,Y 318.741,Z 340.57,A -85,B 0,C 180,E1 -15550.184,E2 -15550.184} C_VEL
LIN {X 0,Y 317.318,Z 351.152,A -85,B 0,C 180,E1 -15551.435,E2 -15551.435} C_VEL
LIN {X 0,Y 316.243,Z 358.899,A -85,B 0,C 180,E1 -15552.542,E2 -15552.542} C_VEL
LIN {X 0,Y 315.151,Z 366.979,A -85,B 0,C 180,E1 -15553.929,E2 -15553.929} C_VEL
LIN {X 0,Y 314.065,Z 374.249,A -85,B 0,C 180,E1 -15555.419,E2 -15555.419} C_VEL
LIN {X 0,Y 312.994,Z 380.787,A -85,B 0,C 180,E1 -15557.024,E2 -15557.024} C_VEL
LIN {X 0,Y 312.325,Z 385.291,A -85,B 0,C 180,E1 -15558.316,E2 -15558.316} C_VEL
LIN {X 0,Y 311.598,Z 390.787,A -85,B 0,C 180,E1 -15560.261,E2 -15560.261} C_VEL
LIN {X 0,Y 311.076,Z 395.115,A -85,B 0,C 180,E1 -15562.209,E2 -15562.209} C_VEL
LIN {X 0,Y 310.911,Z 397.485,A -85,B 0,C 180,E1 -15563.511,E2 -15563.511} C_VEL
LIN {X 0,Y 310.764,Z 399.286,A -85,B 0,C 180,E1 -15564.81,E2 -15564.81} C_VEL
LIN {X 0,Y 310.692,Z 401.737,A -85,B 0,C 180,E1 -15567.407,E2 -15567.407} C_VEL
LIN {X 0,Y 310.652,Z 402.326,A -85,B 0,C 180,E1 -15568.704,E2 -15568.704} C_VEL
LIN {X 0,Y 310.652,Z 402.326,A -85,B 0,C 180,E1 -15571.296,E2 -15571.296} C_VEL
LIN {X 0,Y 310.692,Z 401.737,A -85,B 0,C 180,E1 -15572.593,E2 -15572.593} C_VEL
LIN {X 0,Y 310.764,Z 399.286,A -85,B 0,C 180,E1 -15575.19,E2 -15575.19} C_VEL
LIN {X 0,Y 310.963,Z 396.333,A -85,B 0,C 180,E1 -15577.14,E2 -15577.14} C_VEL
LIN {X 0,Y 311.411,Z 392.342,A -85,B 0,C 180,E1 -15579.089,E2 -15579.089} C_VEL
LIN {X 0,Y 312.066,Z 387.208,A -85,B 0,C 180,E1 -15581.036,E2 -15581.036} C_VEL
LIN {X 0,Y 312.782,Z 381.942,A -85,B 0,C 180,E1 -15582.655,E2 -15582.655} C_VEL
LIN {X 0,Y 313.823,Z 375.625,A -85,B 0,C 180,E1 -15584.261,E2 -15584.261} C_VEL
LIN {X 0,Y 314.683,Z 369.67,A -85,B 0,C 180,E1 -15585.545,E2 -15585.545} C_VEL
LIN {X 0,Y 315.692,Z 362.74,A -85,B 0,C 180,E1 -15586.822,E2 -15586.822} C_VEL
LIN {X 0,Y 316.812,Z 354.556,A -85,B 0,C 180,E1 -15588.093,E2 -15588.093} C_VEL
LIN {X 0,Y 318.039,Z 346.045,A -85,B 0,C 180,E1 -15589.19,E2 -15589.19} C_VEL
LIN {X 0,Y 318.762,Z 340.571,A -85,B 0,C 180,E1 -15589.815,E2 -15589.815} C_VEL
LIN {X 0,Y 317.726,Z 329.488,A -85,B 0,C 180,E1 -15590.983,E2 -15590.983} C_VEL
LIN {X 0,Y 316.199,Z 318.817,A -85,B 0,C 180,E1 -15591.929,E2 -15591.929} C_VEL
LIN {X 0,Y 314.078,Z 308.274,A -85,B 0,C 180,E1 -15592.721,E2 -15592.721} C_VEL
LIN {X 0,Y 311.376,Z 297.688,A -85,B 0,C 180,E1 -15593.384,E2 -15593.384} C_VEL
LIN {X 0,Y 311.297,Z 297.009,A -85,B 0,C 180,E1 -15593.429,E2 -15593.429} C_VEL
LIN {X 0,Y 311.667,Z 293.158,A -85,B 0,C 180,E1 -15596.807,E2 -15596.807} C_VEL
LIN {X 0,Y 312.064,Z 289.943,A -85,B 0,C 180,E1 -15599.7,E2 -15599.7} C_VEL
LIN {X 0,Y 312.643,Z 285.655,A -85,B 0,C 180,E1 -15603.715,E2 -15603.715} C_VEL
LIN {X 0,Y 313.173,Z 282.007,A -85,B 0,C 180,E1 -15607.294,E2 -15607.294} C_VEL
LIN {X 0,Y 313.617,Z 278.884,A -85,B 0,C 180,E1 -15610.531,E2 -15610.531} C_VEL
LIN {X 0,Y 313.746,Z 277.238,A -85,B 0,C 180,E1 -15612.329,E2 -15612.329} C_VEL
LIN {X 0,Y 313.529,Z 274.248,A -85,B 0,C 180,E1 -15615.831,E2 -15615.831} C_VEL
LIN {X 0,Y 313.135,Z 271.505,A -85,B 0,C 180,E1 -15619.386,E2 -15619.386} C_VEL
LIN {X 0,Y 312.798,Z 269.235,A -85,B 0,C 180,E1 -15622.646,E2 -15622.646} C_VEL
LIN {X 0,Y 312.55,Z 267.162,A -85,B 0,C 180,E1 -15625.789,E2 -15625.789} C_VEL
LIN {X 0,Y 312.516,Z 267.058,A -85,B 0,C 180,E1 -15628.846,E2 -15628.846} C_VEL
LIN {X 0,Y 312.516,Z 267.056,A -85,B 0,C 180,E1 -15631.812,E2 -15631.812} C_VEL
LIN {X 0,Y 312.524,Z 267.058,A -85,B 0,C 180,E1 -15634.699,E2 -15634.699} C_VEL
LIN {X 0,Y 312.546,Z 267.053,A -85,B 0,C 180,E1 -15637.519,E2 -15637.519} C_VEL
LIN {X 0,Y 312.551,Z 267.051,A -85,B 0,C 180,E1 -15641.644,E2 -15641.644} C_VEL
LIN {X 0,Y 312.654,Z 267.039,A -85,B 0,C 180,E1 -15645.678,E2 -15645.678} C_VEL
LIN {X 0,Y 312.686,Z 267.035,A -85,B 0,C 180,E1 -15649.634,E2 -15649.634} C_VEL
LIN {X 0,Y 312.794,Z 267.022,A -85,B 0,C 180,E1 -15652.245,E2 -15652.245} C_VEL
LIN {X 0,Y 312.682,Z 267.033,A -85,B 0,C 180,E1 -15654.835,E2 -15654.835} C_VEL
LIN {X 0,Y 312.974,Z 266.996,A -85,B 0,C 180,E1 -15658.706,E2 -15658.706} C_VEL
LIN {X 0,Y 312.903,Z 266.998,A -85,B 0,C 180,E1 -15662.567,E2 -15662.567} C_VEL
LIN {X 0,Y 312.839,Z 267.013,A -85,B 0,C 180,E1 -15666.549,E2 -15666.549} C_VEL
LIN {X 0,Y 312.738,Z 267.028,A -85,B 0,C 180,E1 -15669.042,E2 -15669.042} C_VEL
LIN {X 0,Y 312.617,Z 267.044,A -85,B 0,C 180,E1 -15672.983,E2 -15672.983} C_VEL
LIN {X 0,Y 312.604,Z 267.044,A -85,B 0,C 180,E1 -15675.643,E2 -15675.643} C_VEL
LIN {X 0,Y 312.539,Z 267.05,A -85,B 0,C 180,E1 -15679.703,E2 -15679.703} C_VEL
LIN {X 0,Y 312.502,Z 267.059,A -85,B 0,C 180,E1 -15682.772,E2 -15682.772} C_VEL
LIN {X 0,Y 312.57,Z 267.046,A -85,B 0,C 180,E1 -15685.925,E2 -15685.925} C_VEL
LIN {X 0,Y 312.508,Z 267.055,A -85,B 0,C 180,E1 -15689.643,E2 -15689.643} C_VEL
LIN {X 0,Y 312.486,Z 267.057,A -85,B 0,C 180,E1 -15693.681,E2 -15693.681} C_VEL
LIN {X 0,Y 312.503,Z 267.056,A -85,B 0,C 180,E1 -15697.376,E2 -15697.376} C_VEL
LIN {X 0,Y 312.488,Z 267.061,A -85,B 0,C 180,E1 -15700.696,E2 -15700.696} C_VEL
LIN {X 0,Y 312.553,Z 267.053,A -85,B 0,C 180,E1 -15704.178,E2 -15704.178} C_VEL
LIN {X 0,Y 312.512,Z 267.056,A -85,B 0,C 180,E1 -15707.898,E2 -15707.898} C_VEL
LIN {X 0,Y 312.496,Z 267.06,A -85,B 0,C 180,E1 -15711.903,E2 -15711.903} C_VEL
LIN {X 0,Y 312.457,Z 267.065,A -85,B 0,C 180,E1 -15715.785,E2 -15715.785} C_VEL
LIN {X 0,Y 312.476,Z 267.06,A -85,B 0,C 180,E1 -15718.849,E2 -15718.849} C_VEL
LIN {X 0,Y 312.522,Z 267.058,A -85,B 0,C 180,E1 -15721.82,E2 -15721.82} C_VEL
LIN {X 0,Y 312.541,Z 267.052,A -85,B 0,C 180,E1 -15724.708,E2 -15724.708} C_VEL
LIN {X 0,Y 312.541,Z 267.079,A -85,B 0,C 180,E1 -15726.357,E2 -15726.357} C_VEL
LIN {X 0,Y 313.557,Z 269.937,A -85,B 0,C 180,E1 -15726.521,E2 -15726.521} C_VEL
LIN {X 0,Y 318.521,Z 277.986,A -85,B 0,C 180,E1 -15727.227,E2 -15727.227} C_VEL
LIN {X 0,Y 323.286,Z 284.384,A -85,B 0,C 180,E1 -15727.988,E2 -15727.988} C_VEL
LIN {X 0,Y 328.139,Z 290.42,A -85,B 0,C 180,E1 -15728.842,E2 -15728.842} C_VEL
LIN {X 0,Y 332.287,Z 295.432,A -85,B 0,C 180,E1 -15729.633,E2 -15729.633} C_VEL
LIN {X 0,Y 337.934,Z 301.856,A -85,B 0,C 180,E1 -15730.806,E2 -15730.806} C_VEL
LIN {X 0,Y 343.66,Z 307.992,A -85,B 0,C 180,E1 -15732.1,E2 -15732.1} C_VEL
LIN {X 0,Y 347.944,Z 312.526,A -85,B 0,C 180,E1 -15733.163,E2 -15733.163} C_VEL
LIN {X 0,Y 352.56,Z 316.579,A -85,B 0,C 180,E1 -15734.345,E2 -15734.345} C_VEL
LIN {X 0,Y 356.935,Z 321.18,A -85,B 0,C 180,E1 -15735.665,E2 -15735.665} C_VEL
LIN {X 0,Y 361.441,Z 325.019,A -85,B 0,C 180,E1 -15737.099,E2 -15737.099} C_VEL
LIN {X 0,Y 365.541,Z 328.902,A -85,B 0,C 180,E1 -15738.628,E2 -15738.628} C_VEL
LIN {X 0,Y 369.423,Z 331.504,A -85,B 0,C 180,E1 -15740.142,E2 -15740.142} C_VEL
LIN {X 0,Y 371.62,Z 333.862,A -85,B 0,C 180,E1 -15741.298,E2 -15741.298} C_VEL
LIN {X 0,Y 373.516,Z 335.802,A -85,B 0,C 180,E1 -15742.432,E2 -15742.432} C_VEL
LIN {X 0,Y 375.287,Z 337.212,A -85,B 0,C 180,E1 -15743.549,E2 -15743.549} C_VEL
LIN {X 0,Y 376.813,Z 338.179,A -85,B 0,C 180,E1 -15744.649,E2 -15744.649} C_VEL
LIN {X 0,Y 378.13,Z 338.782,A -85,B 0,C 180,E1 -15745.737,E2 -15745.737} C_VEL
LIN {X 0,Y 379.795,Z 339.216,A -85,B 0,C 180,E1 -15747.549,E2 -15747.549} C_VEL
LIN {X 0,Y 380.518,Z 339.33,A -85,B 0,C 180,E1 -15748.942,E2 -15748.942} C_VEL
LIN {X 0,Y 380.677,Z 339.36,A -85,B 0,C 180,E1 -15750,E2 -15750} C_VEL
LIN {X 0,Y 380.513,Z 339.315,A -85,B 0,C 180,E1 -15751.058,E2 -15751.058} C_VEL
LIN {X 0,Y 379.795,Z 339.22,A -85,B 0,C 180,E1 -15752.451,E2 -15752.451} C_VEL
LIN {X 0,Y 378.137,Z 338.794,A -85,B 0,C 180,E1 -15754.263,E2 -15754.263} C_VEL
LIN {X 0,Y 376.831,Z 338.183,A -85,B 0,C 180,E1 -15755.351,E2 -15755.351} C_VEL
LIN {X 0,Y 374.955,Z 336.962,A -85,B 0,C 180,E1 -15756.666,E2 -15756.666} C_VEL
LIN {X 0,Y 373.54,Z 335.81,A -85,B 0,C 180,E1 -15757.568,E2 -15757.568} C_VEL
LIN {X 0,Y 370.359,Z 332.457,A -85,B 0,C 180,E1 -15759.393,E2 -15759.393} C_VEL
LIN {X 0,Y 369.432,Z 331.507,A -85,B 0,C 180,E1 -15759.858,E2 -15759.858} C_VEL
LIN {X 0,Y 365.531,Z 328.914,A -85,B 0,C 180,E1 -15761.364,E2 -15761.364} C_VEL
LIN {X 0,Y 363.094,Z 326.767,A -85,B 0,C 180,E1 -15762.293,E2 -15762.293} C_VEL
LIN {X 0,Y 358.266,Z 322.269,A -85,B 0,C 180,E1 -15763.922,E2 -15763.922} C_VEL
LIN {X 0,Y 354.987,Z 319.318,A -85,B 0,C 180,E1 -15764.914,E2 -15764.914} C_VEL
LIN {X 0,Y 350.973,Z 315.28,A -85,B 0,C 180,E1 -15766.056,E2 -15766.056} C_VEL
LIN {X 0,Y 346.503,Z 310.945,A -85,B 0,C 180,E1 -15767.203,E2 -15767.203} C_VEL
LIN {X 0,Y 340.006,Z 304.183,A -85,B 0,C 180,E1 -15768.733,E2 -15768.733} C_VEL
LIN {X 0,Y 333.75,Z 297.144,A -85,B 0,C 180,E1 -15770.07,E2 -15770.07} C_VEL
LIN {X 0,Y 328.666,Z 291.097,A -85,B 0,C 180,E1 -15771.056,E2 -15771.056} C_VEL
LIN {X 0,Y 324.418,Z 285.794,A -85,B 0,C 180,E1 -15771.821,E2 -15771.821} C_VEL
LIN {X 0,Y 320.397,Z 280.562,A -85,B 0,C 180,E1 -15772.485,E2 -15772.485} C_VEL
LIN {X 0,Y 316.838,Z 275.251,A -85,B 0,C 180,E1 -15773.022,E2 -15773.022} C_VEL
LIN {X 0,Y 314.52,Z 271.434,A -85,B 0,C 180,E1 -15773.355,E2 -15773.355} C_VEL
LIN {X 0,Y 312.76,Z 268.115,A -85,B 0,C 180,E1 -15773.597,E2 -15773.597} C_VEL
LIN {X 0,Y 312.524,Z 267.056,A -85,B 0,C 180,E1 -15773.648,E2 -15773.648} C_VEL
LIN {X 0,Y 312.502,Z 267.058,A -85,B 0,C 180,E1 -15776.73,E2 -15776.73} C_VEL
LIN {X 0,Y 312.494,Z 267.059,A -85,B 0,C 180,E1 -15779.655,E2 -15779.655} C_VEL
LIN {X 0,Y 312.47,Z 267.063,A -85,B 0,C 180,E1 -15783.694,E2 -15783.694} C_VEL
LIN {X 0,Y 312.492,Z 267.059,A -85,B 0,C 180,E1 -15787.389,E2 -15787.389} C_VEL
LIN {X 0,Y 312.483,Z 267.058,A -85,B 0,C 180,E1 -15790.709,E2 -15790.709} C_VEL
LIN {X 0,Y 312.552,Z 267.051,A -85,B 0,C 180,E1 -15794.191,E2 -15794.191} C_VEL
LIN {X 0,Y 312.516,Z 267.057,A -85,B 0,C 180,E1 -15797.911,E2 -15797.911} C_VEL
LIN {X 0,Y 312.506,Z 267.057,A -85,B 0,C 180,E1 -15801.916,E2 -15801.916} C_VEL
LIN {X 0,Y 312.473,Z 267.061,A -85,B 0,C 180,E1 -15805.797,E2 -15805.797} C_VEL
LIN {X 0,Y 312.489,Z 267.06,A -85,B 0,C 180,E1 -15808.861,E2 -15808.861} C_VEL
LIN {X 0,Y 312.541,Z 267.051,A -85,B 0,C 180,E1 -15811.832,E2 -15811.832} C_VEL
LIN {X 0,Y 312.559,Z 267.05,A -85,B 0,C 180,E1 -15814.719,E2 -15814.719} C_VEL
LIN {X 0,Y 312.541,Z 267.052,A -85,B 0,C 180,E1 -15817.535,E2 -15817.535} C_VEL
LIN {X 0,Y 312.562,Z 267.048,A -85,B 0,C 180,E1 -15821.661,E2 -15821.661} C_VEL
LIN {X 0,Y 312.668,Z 267.034,A -85,B 0,C 180,E1 -15825.694,E2 -15825.694} C_VEL
LIN {X 0,Y 312.671,Z 267.033,A -85,B 0,C 180,E1 -15829.649,E2 -15829.649} C_VEL
LIN {X 0,Y 312.817,Z 267.019,A -85,B 0,C 180,E1 -15832.261,E2 -15832.261} C_VEL
LIN {X 0,Y 312.69,Z 267.032,A -85,B 0,C 180,E1 -15834.85,E2 -15834.85} C_VEL
LIN {X 0,Y 312.68,Z 267.032,A -85,B 0,C 180,E1 -15836.298,E2 -15836.298} C_VEL
LIN {X 0,Y 312.153,Z 267.092,A -85,B 0,C 180,E1 -15837.375,E2 -15837.375} C_VEL
LIN {X 0,Y 309.436,Z 267.432,A -85,B 0,C 180,E1 -15839.132,E2 -15839.132} C_VEL
LIN {X 0,Y 307.04,Z 267.738,A -85,B 0,C 180,E1 -15840.556,E2 -15840.556} C_VEL
LIN {X 0,Y 305.974,Z 267.868,A -85,B 0,C 180,E1 -15841.657,E2 -15841.657} C_VEL
LIN {X 0,Y 305.871,Z 267.88,A -85,B 0,C 180,E1 -15842.03,E2 -15842.03} C_VEL
LIN {X 0,Y 305.782,Z 267.895,A -85,B 0,C 180,E1 -15846.606,E2 -15846.606} C_VEL
LIN {X 0,Y 305.695,Z 267.904,A -85,B 0,C 180,E1 -15849.268,E2 -15849.268} C_VEL
LIN {X 0,Y 305.573,Z 267.92,A -85,B 0,C 180,E1 -15853.304,E2 -15853.304} C_VEL
LIN {X 0,Y 305.517,Z 267.93,A -85,B 0,C 180,E1 -15856.031,E2 -15856.031} C_VEL
LIN {X 0,Y 305.482,Z 267.932,A -85,B 0,C 180,E1 -15860.194,E2 -15860.194} C_VEL
LIN {X 0,Y 305.447,Z 267.935,A -85,B 0,C 180,E1 -15864.473,E2 -15864.473} C_VEL
LIN {X 0,Y 305.449,Z 267.939,A -85,B 0,C 180,E1 -15867.405,E2 -15867.405} C_VEL
LIN {X 0,Y 305.427,Z 267.94,A -85,B 0,C 180,E1 -15870.42,E2 -15870.42} C_VEL
LIN {X 0,Y 305.484,Z 267.936,A -85,B 0,C 180,E1 -15873.521,E2 -15873.521} C_VEL
LIN {X 0,Y 305.729,Z 269.889,A -85,B 0,C 180,E1 -15876.711,E2 -15876.711} C_VEL
LIN {X 0,Y 306.134,Z 272.686,A -85,B 0,C 180,E1 -15880.749,E2 -15880.749} C_VEL
LIN {X 0,Y 306.523,Z 275.71,A -85,B 0,C 180,E1 -15884.703,E2 -15884.703} C_VEL
LIN {X 0,Y 306.684,Z 277.755,A -85,B 0,C 180,E1 -15887.172,E2 -15887.172} C_VEL
LIN {X 0,Y 306.479,Z 280.329,A -85,B 0,C 180,E1 -15890.054,E2 -15890.054} C_VEL
LIN {X 0,Y 305.968,Z 283.632,A -85,B 0,C 180,E1 -15893.516,E2 -15893.516} C_VEL
LIN {X 0,Y 305.534,Z 286.612,A -85,B 0,C 180,E1 -15896.493,E2 -15896.493} C_VEL
LIN {X 0,Y 305.066,Z 289.798,A -85,B 0,C 180,E1 -15899.548,E2 -15899.548} C_VEL
LIN {X 0,Y 304.674,Z 293.025,A -85,B 0,C 180,E1 -15902.527,E2 -15902.527} C_VEL
LIN {X 0,Y 304.283,Z 296.822,A -85,B 0,C 180,E1 -15906.006,E2 -15906.006} C_VEL
LIN {X 0,Y 306.726,Z 306.799,A -85,B 0,C 180,E1 -15906.639,E2 -15906.639} C_VEL
LIN {X 0,Y 308.868,Z 316.436,A -85,B 0,C 180,E1 -15907.376,E2 -15907.376} C_VEL
LIN {X 0,Y 310.345,Z 325.964,A -85,B 0,C 180,E1 -15908.21,E2 -15908.21} C_VEL
LIN {X 0,Y 311.434,Z 335.445,A -85,B 0,C 180,E1 -15909.181,E2 -15909.181} C_VEL
LIN {X 0,Y 311.897,Z 341.778,A -85,B 0,C 180,E1 -15909.902,E2 -15909.902} C_VEL
LIN {X 0,Y 310.393,Z 352.074,A -85,B 0,C 180,E1 -15911.177,E2 -15911.177} C_VEL
LIN {X 0,Y 309.136,Z 360.607,A -85,B 0,C 180,E1 -15912.469,E2 -15912.469} C_VEL
LIN {X 0,Y 308.056,Z 368.267,A -85,B 0,C 180,E1 -15913.863,E2 -15913.863} C_VEL
LIN {X 0,Y 306.916,Z 375.412,A -85,B 0,C 180,E1 -15915.411,E2 -15915.411} C_VEL
LIN {X 0,Y 305.84,Z 381.73,A -85,B 0,C 180,E1 -15917.053,E2 -15917.053} C_VEL
LIN {X 0,Y 305.072,Z 386.996,A -85,B 0,C 180,E1 -15918.708,E2 -15918.708} C_VEL
LIN {X 0,Y 304.361,Z 392.129,A -85,B 0,C 180,E1 -15920.698,E2 -15920.698} C_VEL
LIN {X 0,Y 303.886,Z 396.121,A -85,B 0,C 180,E1 -15922.692,E2 -15922.692} C_VEL
LIN {X 0,Y 303.687,Z 399.075,A -85,B 0,C 180,E1 -15924.689,E2 -15924.689} C_VEL
LIN {X 0,Y 303.618,Z 401.526,A -85,B 0,C 180,E1 -15927.347,E2 -15927.347} C_VEL
LIN {X 0,Y 303.57,Z 402.115,A -85,B 0,C 180,E1 -15928.673,E2 -15928.673} C_VEL
LIN {X 0,Y 303.57,Z 402.115,A -85,B 0,C 180,E1 -15931.327,E2 -15931.327} C_VEL
LIN {X 0,Y 303.618,Z 401.526,A -85,B 0,C 180,E1 -15932.653,E2 -15932.653} C_VEL
LIN {X 0,Y 303.687,Z 399.075,A -85,B 0,C 180,E1 -15935.311,E2 -15935.311} C_VEL
LIN {X 0,Y 303.886,Z 396.121,A -85,B 0,C 180,E1 -15937.308,E2 -15937.308} C_VEL
LIN {X 0,Y 304.361,Z 392.129,A -85,B 0,C 180,E1 -15939.302,E2 -15939.302} C_VEL
LIN {X 0,Y 305.071,Z 386.996,A -85,B 0,C 180,E1 -15941.292,E2 -15941.292} C_VEL
LIN {X 0,Y 305.832,Z 381.73,A -85,B 0,C 180,E1 -15942.947,E2 -15942.947} C_VEL
LIN {X 0,Y 306.904,Z 375.412,A -85,B 0,C 180,E1 -15944.589,E2 -15944.589} C_VEL
LIN {X 0,Y 308.053,Z 368.279,A -85,B 0,C 180,E1 -15946.135,E2 -15946.135} C_VEL
LIN {X 0,Y 309.148,Z 360.607,A -85,B 0,C 180,E1 -15947.53,E2 -15947.53} C_VEL
LIN {X 0,Y 310.381,Z 352.074,A -85,B 0,C 180,E1 -15948.824,E2 -15948.824} C_VEL
LIN {X 0,Y 311.907,Z 341.778,A -85,B 0,C 180,E1 -15950.097,E2 -15950.097} C_VEL
LIN {X 0,Y 310.906,Z 330.256,A -85,B 0,C 180,E1 -15951.381,E2 -15951.381} C_VEL
LIN {X 0,Y 309.358,Z 319.065,A -85,B 0,C 180,E1 -15952.408,E2 -15952.408} C_VEL
LIN {X 0,Y 307.168,Z 308.457,A -85,B 0,C 180,E1 -15953.241,E2 -15953.241} C_VEL
LIN {X 0,Y 304.334,Z 297.496,A -85,B 0,C 180,E1 -15953.957,E2 -15953.957} C_VEL
LIN {X 0,Y 304.265,Z 296.812,A -85,B 0,C 180,E1 -15954.005,E2 -15954.005} C_VEL
LIN {X 0,Y 304.671,Z 292.978,A -85,B 0,C 180,E1 -15957.474,E2 -15957.474} C_VEL
LIN {X 0,Y 305.245,Z 288.608,A -85,B 0,C 180,E1 -15961.573,E2 -15961.573} C_VEL
LIN {X 0,Y 305.788,Z 285.022,A -85,B 0,C 180,E1 -15965.07,E2 -15965.07} C_VEL
LIN {X 0,Y 306.337,Z 281.46,A -85,B 0,C 180,E1 -15968.729,E2 -15968.729} C_VEL
LIN {X 0,Y 306.651,Z 278.775,A -85,B 0,C 180,E1 -15971.654,E2 -15971.654} C_VEL
LIN {X 0,Y 306.582,Z 276.172,A -85,B 0,C 180,E1 -15974.706,E2 -15974.706} C_VEL
LIN {X 0,Y 306.236,Z 273.392,A -85,B 0,C 180,E1 -15978.269,E2 -15978.269} C_VEL
LIN {X 0,Y 305.873,Z 270.981,A -85,B 0,C 180,E1 -15981.65,E2 -15981.65} C_VEL
LIN {X 0,Y 305.605,Z 268.87,A -85,B 0,C 180,E1 -15984.899,E2 -15984.899} C_VEL
LIN {X 0,Y 305.484,Z 267.936,A -85,B 0,C 180,E1 -15986.479,E2 -15986.479} C_VEL
LIN {X 0,Y 305.427,Z 267.939,A -85,B 0,C 180,E1 -15989.58,E2 -15989.58} C_VEL
LIN {X 0,Y 305.449,Z 267.94,A -85,B 0,C 180,E1 -15992.595,E2 -15992.595} C_VEL
LIN {X 0,Y 305.447,Z 267.937,A -85,B 0,C 180,E1 -15995.527,E2 -15995.527} C_VEL
LIN {X 0,Y 305.482,Z 267.934,A -85,B 0,C 180,E1 -15999.806,E2 -15999.806} C_VEL
LIN {X 0,Y 305.517,Z 267.93,A -85,B 0,C 180,E1 -16003.969,E2 -16003.969} C_VEL
LIN {X 0,Y 305.573,Z 267.92,A -85,B 0,C 180,E1 -16006.696,E2 -16006.696} C_VEL
LIN {X 0,Y 305.753,Z 267.897,A -85,B 0,C 180,E1 -16011.255,E2 -16011.255} C_VEL
LIN {X 0,Y 305.782,Z 267.894,A -85,B 0,C 180,E1 -16013.394,E2 -16013.394} C_VEL
LIN {X 0,Y 305.941,Z 267.872,A -85,B 0,C 180,E1 -16018.676,E2 -16018.676} C_VEL
LIN {X 0,Y 305.929,Z 267.871,A -85,B 0,C 180,E1 -16021.309,E2 -16021.309} C_VEL
LIN {X 0,Y 305.66,Z 267.908,A -85,B 0,C 180,E1 -16025.269,E2 -16025.269} C_VEL
LIN {X 0,Y 305.758,Z 267.897,A -85,B 0,C 180,E1 -16027.919,E2 -16027.919} C_VEL
LIN {X 0,Y 305.582,Z 267.919,A -85,B 0,C 180,E1 -16031.937,E2 -16031.937} C_VEL
LIN {X 0,Y 305.591,Z 267.919,A -85,B 0,C 180,E1 -16035.006,E2 -16035.006} C_VEL
LIN {X 0,Y 305.522,Z 267.925,A -85,B 0,C 180,E1 -16039.418,E2 -16039.418} C_VEL
LIN {X 0,Y 305.463,Z 267.937,A -85,B 0,C 180,E1 -16043.031,E2 -16043.031} C_VEL
LIN {X 0,Y 305.499,Z 267.928,A -85,B 0,C 180,E1 -16046.21,E2 -16046.21} C_VEL
LIN {X 0,Y 305.459,Z 267.937,A -85,B 0,C 180,E1 -16049.039,E2 -16049.039} C_VEL
LIN {X 0,Y 305.41,Z 267.939,A -85,B 0,C 180,E1 -16051.945,E2 -16051.945} C_VEL
LIN {X 0,Y 305.427,Z 267.938,A -85,B 0,C 180,E1 -16055.106,E2 -16055.106} C_VEL
LIN {X 0,Y 305.445,Z 267.939,A -85,B 0,C 180,E1 -16058.529,E2 -16058.529} C_VEL
LIN {X 0,Y 305.481,Z 267.934,A -85,B 0,C 180,E1 -16062.592,E2 -16062.592} C_VEL
LIN {X 0,Y 305.491,Z 267.934,A -85,B 0,C 180,E1 -16066.358,E2 -16066.358} C_VEL
LIN {X 0,Y 305.439,Z 267.938,A -85,B 0,C 180,E1 -16069.89,E2 -16069.89} C_VEL
LIN {X 0,Y 305.436,Z 267.938,A -85,B 0,C 180,E1 -16073.625,E2 -16073.625} C_VEL
LIN {X 0,Y 305.416,Z 267.941,A -85,B 0,C 180,E1 -16076.478,E2 -16076.478} C_VEL
LIN {X 0,Y 305.414,Z 267.942,A -85,B 0,C 180,E1 -16079.586,E2 -16079.586} C_VEL
LIN {X 0,Y 305.469,Z 267.933,A -85,B 0,C 180,E1 -16082.604,E2 -16082.604} C_VEL
LIN {X 0,Y 305.479,Z 267.935,A -85,B 0,C 180,E1 -16085.745,E2 -16085.745} C_VEL
LIN {X 0,Y 306.488,Z 270.763,A -85,B 0,C 180,E1 -16085.919,E2 -16085.919} C_VEL
LIN {X 0,Y 310.96,Z 278.733,A -85,B 0,C 180,E1 -16086.513,E2 -16086.513} C_VEL
LIN {X 0,Y 316.634,Z 287.055,A -85,B 0,C 180,E1 -16087.373,E2 -16087.373} C_VEL
LIN {X 0,Y 323.228,Z 295.22,A -85,B 0,C 180,E1 -16088.494,E2 -16088.494} C_VEL
LIN {X 0,Y 328.123,Z 301.03,A -85,B 0,C 180,E1 -16089.426,E2 -16089.426} C_VEL
LIN {X 0,Y 333.127,Z 306.844,A -85,B 0,C 180,E1 -16090.476,E2 -16090.476} C_VEL
LIN {X 0,Y 339.887,Z 313.966,A -85,B 0,C 180,E1 -16091.986,E2 -16091.986} C_VEL
LIN {X 0,Y 345.677,Z 319.938,A -85,B 0,C 180,E1 -16093.463,E2 -16093.463} C_VEL
LIN {X 0,Y 349.841,Z 323.856,A -85,B 0,C 180,E1 -16094.601,E2 -16094.601} C_VEL
LIN {X 0,Y 352.777,Z 326.843,A -85,B 0,C 180,E1 -16095.492,E2 -16095.492} C_VEL
LIN {X 0,Y 357.384,Z 330.758,A -85,B 0,C 180,E1 -16096.95,E2 -16096.95} C_VEL
LIN {X 0,Y 361.45,Z 334.631,A -85,B 0,C 180,E1 -16098.461,E2 -16098.461} C_VEL
LIN {X 0,Y 365.534,Z 337.433,A -85,B 0,C 180,E1 -16100.036,E2 -16100.036} C_VEL
LIN {X 0,Y 369.023,Z 341.072,A -85,B 0,C 180,E1 -16101.956,E2 -16101.956} C_VEL
LIN {X 0,Y 371.427,Z 343.142,A -85,B 0,C 180,E1 -16103.481,E2 -16103.481} C_VEL
LIN {X 0,Y 373.737,Z 344.522,A -85,B 0,C 180,E1 -16105.189,E2 -16105.189} C_VEL
LIN {X 0,Y 375.441,Z 345.092,A -85,B 0,C 180,E1 -16106.781,E2 -16106.781} C_VEL
LIN {X 0,Y 376.266,Z 345.303,A -85,B 0,C 180,E1 -16107.859,E2 -16107.859} C_VEL
LIN {X 0,Y 376.803,Z 345.371,A -85,B 0,C 180,E1 -16108.931,E2 -16108.931} C_VEL
LIN {X 0,Y 376.97,Z 345.404,A -85,B 0,C 180,E1 -16110,E2 -16110} C_VEL
LIN {X 0,Y 376.794,Z 345.363,A -85,B 0,C 180,E1 -16111.069,E2 -16111.069} C_VEL
LIN {X 0,Y 376.261,Z 345.286,A -85,B 0,C 180,E1 -16112.141,E2 -16112.141} C_VEL
LIN {X 0,Y 375.439,Z 345.073,A -85,B 0,C 180,E1 -16113.219,E2 -16113.219} C_VEL
LIN {X 0,Y 373.735,Z 344.505,A -85,B 0,C 180,E1 -16114.807,E2 -16114.807} C_VEL
LIN {X 0,Y 371.396,Z 343.156,A -85,B 0,C 180,E1 -16116.519,E2 -16116.519} C_VEL
LIN {X 0,Y 369.025,Z 341.072,A -85,B 0,C 180,E1 -16118.046,E2 -16118.046} C_VEL
LIN {X 0,Y 365.533,Z 337.442,A -85,B 0,C 180,E1 -16119.964,E2 -16119.964} C_VEL
LIN {X 0,Y 361.413,Z 334.634,A -85,B 0,C 180,E1 -16121.543,E2 -16121.543} C_VEL
LIN {X 0,Y 357.331,Z 330.755,A -85,B 0,C 180,E1 -16123.059,E2 -16123.059} C_VEL
LIN {X 0,Y 352.729,Z 326.833,A -85,B 0,C 180,E1 -16124.51,E2 -16124.51} C_VEL
LIN {X 0,Y 346.858,Z 320.967,A -85,B 0,C 180,E1 -16126.239,E2 -16126.239} C_VEL
LIN {X 0,Y 341.829,Z 315.956,A -85,B 0,C 180,E1 -16127.536,E2 -16127.536} C_VEL
LIN {X 0,Y 336.703,Z 310.744,A -85,B 0,C 180,E1 -16128.741,E2 -16128.741} C_VEL
LIN {X 0,Y 329.595,Z 302.803,A -85,B 0,C 180,E1 -16130.276,E2 -16130.276} C_VEL
LIN {X 0,Y 323.906,Z 296.058,A -85,B 0,C 180,E1 -16131.375,E2 -16131.375} C_VEL
LIN {X 0,Y 319.531,Z 290.567,A -85,B 0,C 180,E1 -16132.162,E2 -16132.162} C_VEL
LIN {X 0,Y 315.43,Z 285.264,A -85,B 0,C 180,E1 -16132.827,E2 -16132.827} C_VEL
LIN {X 0,Y 310.231,Z 277.606,A -85,B 0,C 180,E1 -16133.587,E2 -16133.587} C_VEL
LIN {X 0,Y 305.888,Z 269.522,A -85,B 0,C 180,E1 -16134.163,E2 -16134.163} C_VEL
LIN {X 0,Y 305.473,Z 267.936,A -85,B 0,C 180,E1 -16134.274,E2 -16134.274} C_VEL
LIN {X 0,Y 305.469,Z 267.933,A -85,B 0,C 180,E1 -16137.396,E2 -16137.396} C_VEL
LIN {X 0,Y 305.414,Z 267.942,A -85,B 0,C 180,E1 -16140.414,E2 -16140.414} C_VEL
LIN {X 0,Y 305.416,Z 267.943,A -85,B 0,C 180,E1 -16144.084,E2 -16144.084} C_VEL
LIN {X 0,Y 305.433,Z 267.937,A -85,B 0,C 180,E1 -16146.744,E2 -16146.744} C_VEL
LIN {X 0,Y 305.441,Z 267.935,A -85,B 0,C 180,E1 -16150.613,E2 -16150.613} C_VEL
LIN {X 0,Y 305.502,Z 267.928,A -85,B 0,C 180,E1 -16154.523,E2 -16154.523} C_VEL
LIN {X 0,Y 305.461,Z 267.934,A -85,B 0,C 180,E1 -16158.16,E2 -16158.16} C_VEL
LIN {X 0,Y 305.471,Z 267.936,A -85,B 0,C 180,E1 -16161.609,E2 -16161.609} C_VEL
LIN {X 0,Y 305.427,Z 267.938,A -85,B 0,C 180,E1 -16164.894,E2 -16164.894} C_VEL
LIN {X 0,Y 305.418,Z 267.938,A -85,B 0,C 180,E1 -16168.364,E2 -16168.364} C_VEL
LIN {X 0,Y 305.484,Z 267.934,A -85,B 0,C 180,E1 -16171.121,E2 -16171.121} C_VEL
LIN {X 0,Y 305.539,Z 267.922,A -85,B 0,C 180,E1 -16174.095,E2 -16174.095} C_VEL
LIN {X 0,Y 305.453,Z 267.935,A -85,B 0,C 180,E1 -16178.409,E2 -16178.409} C_VEL
LIN {X 0,Y 305.523,Z 267.927,A -85,B 0,C 180,E1 -16181.223,E2 -16181.223} C_VEL
LIN {X 0,Y 305.609,Z 267.914,A -85,B 0,C 180,E1 -16185.356,E2 -16185.356} C_VEL
LIN {X 0,Y 305.61,Z 267.913,A -85,B 0,C 180,E1 -16189.407,E2 -16189.407} C_VEL
LIN {X 0,Y 305.758,Z 267.897,A -85,B 0,C 180,E1 -16192.081,E2 -16192.081} C_VEL
LIN {X 0,Y 305.66,Z 267.908,A -85,B 0,C 180,E1 -16194.731,E2 -16194.731} C_VEL
LIN {X 0,Y 305.929,Z 267.871,A -85,B 0,C 180,E1 -16198.691,E2 -16198.691} C_VEL
LIN {X 0,Y 305.871,Z 267.88,A -85,B 0,C 180,E1 -16202.03,E2 -16202.03} C_VEL
LIN {X 0,Y 305.147,Z 267.973,A -85,B 0,C 180,E1 -16203.128,E2 -16203.128} C_VEL
LIN {X 0,Y 302.233,Z 268.336,A -85,B 0,C 180,E1 -16204.913,E2 -16204.913} C_VEL
LIN {X 0,Y 299.797,Z 268.642,A -85,B 0,C 180,E1 -16206.361,E2 -16206.361} C_VEL
LIN {X 0,Y 298.767,Z 268.768,A -85,B 0,C 180,E1 -16207.483,E2 -16207.483} C_VEL
LIN {X 0,Y 298.69,Z 268.779,A -85,B 0,C 180,E1 -16207.863,E2 -16207.863} C_VEL
LIN {X 0,Y 298.546,Z 268.798,A -85,B 0,C 180,E1 -16212.239,E2 -16212.239} C_VEL
LIN {X 0,Y 298.528,Z 268.798,A -85,B 0,C 180,E1 -16215.157,E2 -16215.157} C_VEL
LIN {X 0,Y 298.438,Z 268.812,A -85,B 0,C 180,E1 -16219.618,E2 -16219.618} C_VEL
LIN {X 0,Y 298.39,Z 268.82,A -85,B 0,C 180,E1 -16223.61,E2 -16223.61} C_VEL
LIN {X 0,Y 298.41,Z 268.812,A -85,B 0,C 180,E1 -16226.589,E2 -16226.589} C_VEL
LIN {X 0,Y 298.367,Z 268.823,A -85,B 0,C 180,E1 -16229.654,E2 -16229.654} C_VEL
LIN {X 0,Y 298.408,Z 268.817,A -85,B 0,C 180,E1 -16232.806,E2 -16232.806} C_VEL
LIN {X 0,Y 298.662,Z 270.568,A -85,B 0,C 180,E1 -16236.043,E2 -16236.043} C_VEL
LIN {X 0,Y 298.961,Z 272.788,A -85,B 0,C 180,E1 -16239.406,E2 -16239.406} C_VEL
LIN {X 0,Y 299.36,Z 275.604,A -85,B 0,C 180,E1 -16243.301,E2 -16243.301} C_VEL
LIN {X 0,Y 299.646,Z 278.253,A -85,B 0,C 180,E1 -16246.65,E2 -16246.65} C_VEL
LIN {X 0,Y 299.543,Z 280.212,A -85,B 0,C 180,E1 -16248.934,E2 -16248.934} C_VEL
LIN {X 0,Y 299.087,Z 283.318,A -85,B 0,C 180,E1 -16252.342,E2 -16252.342} C_VEL
LIN {X 0,Y 298.601,Z 286.466,A -85,B 0,C 180,E1 -16255.607,E2 -16255.607} C_VEL
LIN {X 0,Y 298.116,Z 289.638,A -85,B 0,C 180,E1 -16258.759,E2 -16258.759} C_VEL
LIN {X 0,Y 297.682,Z 292.826,A -85,B 0,C 180,E1 -16261.825,E2 -16261.825} C_VEL
LIN {X 0,Y 297.246,Z 296.813,A -85,B 0,C 180,E1 -16265.418,E2 -16265.418} C_VEL
LIN {X 0,Y 299.733,Z 306.576,A -85,B 0,C 180,E1 -16266.061,E2 -16266.061} C_VEL
LIN {X 0,Y 301.969,Z 316.367,A -85,B 0,C 180,E1 -16266.84,E2 -16266.84} C_VEL
LIN {X 0,Y 303.349,Z 324.978,A -85,B 0,C 180,E1 -16267.613,E2 -16267.613} C_VEL
LIN {X 0,Y 304.405,Z 333.582,A -85,B 0,C 180,E1 -16268.499,E2 -16268.499} C_VEL
LIN {X 0,Y 305.034,Z 342.918,A -85,B 0,C 180,E1 -16269.606,E2 -16269.606} C_VEL
LIN {X 0,Y 303.688,Z 351.863,A -85,B 0,C 180,E1 -16270.745,E2 -16270.745} C_VEL
LIN {X 0,Y 302.34,Z 360.394,A -85,B 0,C 180,E1 -16272.062,E2 -16272.062} C_VEL
LIN {X 0,Y 301.315,Z 367.579,A -85,B 0,C 180,E1 -16273.39,E2 -16273.39} C_VEL
LIN {X 0,Y 300.262,Z 373.824,A -85,B 0,C 180,E1 -16274.733,E2 -16274.733} C_VEL
LIN {X 0,Y 299.126,Z 380.363,A -85,B 0,C 180,E1 -16276.412,E2 -16276.412} C_VEL
LIN {X 0,Y 298.345,Z 384.865,A -85,B 0,C 180,E1 -16277.76,E2 -16277.76} C_VEL
LIN {X 0,Y 297.536,Z 390.362,A -85,B 0,C 180,E1 -16279.796,E2 -16279.796} C_VEL
LIN {X 0,Y 296.984,Z 394.691,A -85,B 0,C 180,E1 -16281.837,E2 -16281.837} C_VEL
LIN {X 0,Y 296.757,Z 397.061,A -85,B 0,C 180,E1 -16283.2,E2 -16283.2} C_VEL
LIN {X 0,Y 296.602,Z 398.863,A -85,B 0,C 180,E1 -16284.561,E2 -16284.561} C_VEL
LIN {X 0,Y 296.545,Z 401.315,A -85,B 0,C 180,E1 -16287.283,E2 -16287.283} C_VEL
LIN {X 0,Y 296.491,Z 401.904,A -85,B 0,C 180,E1 -16288.642,E2 -16288.642} C_VEL
LIN {X 0,Y 296.491,Z 401.904,A -85,B 0,C 180,E1 -16291.358,E2 -16291.358} C_VEL
LIN {X 0,Y 296.545,Z 401.315,A -85,B 0,C 180,E1 -16292.717,E2 -16292.717} C_VEL
LIN {X 0,Y 296.622,Z 398.863,A -85,B 0,C 180,E1 -16295.438,E2 -16295.438} C_VEL
LIN {X 0,Y 296.834,Z 395.909,A -85,B 0,C 180,E1 -16297.482,E2 -16297.482} C_VEL
LIN {X 0,Y 297.328,Z 391.917,A -85,B 0,C 180,E1 -16299.524,E2 -16299.524} C_VEL
LIN {X 0,Y 298.059,Z 386.783,A -85,B 0,C 180,E1 -16301.561,E2 -16301.561} C_VEL
LIN {X 0,Y 298.903,Z 381.518,A -85,B 0,C 180,E1 -16303.253,E2 -16303.253} C_VEL
LIN {X 0,Y 300,Z 375.2,A -85,B 0,C 180,E1 -16304.933,E2 -16304.933} C_VEL
LIN {X 0,Y 301.01,Z 369.247,A -85,B 0,C 180,E1 -16306.27,E2 -16306.27} C_VEL
LIN {X 0,Y 302.056,Z 362.315,A -85,B 0,C 180,E1 -16307.606,E2 -16307.606} C_VEL
LIN {X 0,Y 303.319,Z 354.132,A -85,B 0,C 180,E1 -16308.928,E2 -16308.928} C_VEL
LIN {X 0,Y 304.65,Z 345.622,A -85,B 0,C 180,E1 -16310.069,E2 -16310.069} C_VEL
LIN {X 0,Y 305.048,Z 341.561,A -85,B 0,C 180,E1 -16310.569,E2 -16310.569} C_VEL
LIN {X 0,Y 304.074,Z 330.371,A -85,B 0,C 180,E1 -16311.856,E2 -16311.856} C_VEL
LIN {X 0,Y 302.442,Z 318.895,A -85,B 0,C 180,E1 -16312.946,E2 -16312.946} C_VEL
LIN {X 0,Y 300.136,Z 308.081,A -85,B 0,C 180,E1 -16313.827,E2 -16313.827} C_VEL
LIN {X 0,Y 297.32,Z 297.457,A -85,B 0,C 180,E1 -16314.553,E2 -16314.553} C_VEL
LIN {X 0,Y 297.241,Z 296.625,A -85,B 0,C 180,E1 -16314.601,E2 -16314.601} C_VEL
LIN {X 0,Y 297.853,Z 291.759,A -85,B 0,C 180,E1 -16319.177,E2 -16319.177} C_VEL
LIN {X 0,Y 298.347,Z 288.029,A -85,B 0,C 180,E1 -16322.805,E2 -16322.805} C_VEL
LIN {X 0,Y 298.859,Z 284.884,A -85,B 0,C 180,E1 -16326.008,E2 -16326.008} C_VEL
LIN {X 0,Y 299.34,Z 281.757,A -85,B 0,C 180,E1 -16329.339,E2 -16329.339} C_VEL
LIN {X 0,Y 299.67,Z 278.652,A -85,B 0,C 180,E1 -16332.852,E2 -16332.852} C_VEL
LIN {X 0,Y 299.507,Z 276.697,A -85,B 0,C 180,E1 -16335.247,E2 -16335.247} C_VEL
LIN {X 0,Y 299.147,Z 273.989,A -85,B 0,C 180,E1 -16338.859,E2 -16338.859} C_VEL
LIN {X 0,Y 298.789,Z 271.636,A -85,B 0,C 180,E1 -16342.29,E2 -16342.29} C_VEL
LIN {X 0,Y 298.554,Z 269.565,A -85,B 0,C 180,E1 -16345.593,E2 -16345.593} C_VEL
LIN {X 0,Y 298.408,Z 268.818,A -85,B 0,C 180,E1 -16347.194,E2 -16347.194} C_VEL
LIN {X 0,Y 298.374,Z 268.821,A -85,B 0,C 180,E1 -16350.633,E2 -16350.633} C_VEL
LIN {X 0,Y 298.42,Z 268.815,A -85,B 0,C 180,E1 -16354.911,E2 -16354.911} C_VEL
LIN {X 0,Y 298.398,Z 268.817,A -85,B 0,C 180,E1 -16357.855,E2 -16357.855} C_VEL
LIN {X 0,Y 298.458,Z 268.808,A -85,B 0,C 180,E1 -16360.744,E2 -16360.744} C_VEL
LIN {X 0,Y 298.514,Z 268.799,A -85,B 0,C 180,E1 -16364.984,E2 -16364.984} C_VEL
LIN {X 0,Y 298.583,Z 268.79,A -85,B 0,C 180,E1 -16369.139,E2 -16369.139} C_VEL
LIN {X 0,Y 298.697,Z 268.78,A -85,B 0,C 180,E1 -16371.877,E2 -16371.877} C_VEL
LIN {X 0,Y 298.623,Z 268.785,A -85,B 0,C 180,E1 -16374.591,E2 -16374.591} C_VEL
LIN {X 0,Y 298.907,Z 268.748,A -85,B 0,C 180,E1 -16378.645,E2 -16378.645} C_VEL
LIN {X 0,Y 298.897,Z 268.745,A -85,B 0,C 180,E1 -16381.339,E2 -16381.339} C_VEL
LIN {X 0,Y 298.742,Z 268.77,A -85,B 0,C 180,E1 -16386.747,E2 -16386.747} C_VEL
LIN {X 0,Y 298.613,Z 268.788,A -85,B 0,C 180,E1 -16389.474,E2 -16389.474} C_VEL
LIN {X 0,Y 298.528,Z 268.797,A -85,B 0,C 180,E1 -16393.608,E2 -16393.608} C_VEL
LIN {X 0,Y 298.468,Z 268.804,A -85,B 0,C 180,E1 -16396.404,E2 -16396.404} C_VEL
LIN {X 0,Y 298.462,Z 268.803,A -85,B 0,C 180,E1 -16399.631,E2 -16399.631} C_VEL
LIN {X 0,Y 298.405,Z 268.812,A -85,B 0,C 180,E1 -16403.592,E2 -16403.592} C_VEL
LIN {X 0,Y 298.459,Z 268.806,A -85,B 0,C 180,E1 -16406.567,E2 -16406.567} C_VEL
LIN {X 0,Y 298.387,Z 268.814,A -85,B 0,C 180,E1 -16409.634,E2 -16409.634} C_VEL
LIN {X 0,Y 298.363,Z 268.821,A -85,B 0,C 180,E1 -16412.793,E2 -16412.793} C_VEL
LIN {X 0,Y 298.43,Z 268.812,A -85,B 0,C 180,E1 -16416.805,E2 -16416.805} C_VEL
LIN {X 0,Y 298.415,Z 268.811,A -85,B 0,C 180,E1 -16421.243,E2 -16421.243} C_VEL
LIN {X 0,Y 298.447,Z 268.807,A -85,B 0,C 180,E1 -16425.054,E2 -16425.054} C_VEL
LIN {X 0,Y 298.409,Z 268.812,A -85,B 0,C 180,E1 -16428.892,E2 -16428.892} C_VEL
LIN {X 0,Y 298.404,Z 268.812,A -85,B 0,C 180,E1 -16433.185,E2 -16433.185} C_VEL
LIN {X 0,Y 298.348,Z 268.82,A -85,B 0,C 180,E1 -16437.195,E2 -16437.195} C_VEL
LIN {X 0,Y 298.381,Z 268.816,A -85,B 0,C 180,E1 -16440.61,E2 -16440.61} C_VEL
LIN {X 0,Y 298.432,Z 268.812,A -85,B 0,C 180,E1 -16443.47,E2 -16443.47} C_VEL
LIN {X 0,Y 298.434,Z 268.811,A -85,B 0,C 180,E1 -16445.15,E2 -16445.15} C_VEL
LIN {X 0,Y 299.562,Z 271.864,A -85,B 0,C 180,E1 -16445.348,E2 -16445.348} C_VEL
LIN {X 0,Y 304.459,Z 281.322,A -85,B 0,C 180,E1 -16446.05,E2 -16446.05} C_VEL
LIN {X 0,Y 309.593,Z 288.95,A -85,B 0,C 180,E1 -16446.808,E2 -16446.808} C_VEL
LIN {X 0,Y 314.007,Z 294.792,A -85,B 0,C 180,E1 -16447.518,E2 -16447.518} C_VEL
LIN {X 0,Y 320.361,Z 302.867,A -85,B 0,C 180,E1 -16448.666,E2 -16448.666} C_VEL
LIN {X 0,Y 327.104,Z 310.636,A -85,B 0,C 180,E1 -16450.02,E2 -16450.02} C_VEL
LIN {X 0,Y 333.535,Z 317.604,A -85,B 0,C 180,E1 -16451.446,E2 -16451.446} C_VEL
LIN {X 0,Y 340.653,Z 324.898,A -85,B 0,C 180,E1 -16453.212,E2 -16453.212} C_VEL
LIN {X 0,Y 345.037,Z 328.924,A -85,B 0,C 180,E1 -16454.381,E2 -16454.381} C_VEL
LIN {X 0,Y 348.47,Z 332.462,A -85,B 0,C 180,E1 -16455.442,E2 -16455.442} C_VEL
LIN {X 0,Y 353.351,Z 336.715,A -85,B 0,C 180,E1 -16457.011,E2 -16457.011} C_VEL
LIN {X 0,Y 358.157,Z 341.045,A -85,B 0,C 180,E1 -16458.801,E2 -16458.801} C_VEL
LIN {X 0,Y 361.063,Z 342.968,A -85,B 0,C 180,E1 -16459.911,E2 -16459.911} C_VEL
LIN {X 0,Y 363.322,Z 345.262,A -85,B 0,C 180,E1 -16461.098,E2 -16461.098} C_VEL
LIN {X 0,Y 365.248,Z 347.254,A -85,B 0,C 180,E1 -16462.259,E2 -16462.259} C_VEL
LIN {X 0,Y 367.556,Z 349.08,A -85,B 0,C 180,E1 -16463.78,E2 -16463.78} C_VEL
LIN {X 0,Y 369.99,Z 350.409,A -85,B 0,C 180,E1 -16465.643,E2 -16465.643} C_VEL
LIN {X 0,Y 371.172,Z 350.801,A -85,B 0,C 180,E1 -16466.744,E2 -16466.744} C_VEL
LIN {X 0,Y 372.515,Z 351.103,A -85,B 0,C 180,E1 -16468.706,E2 -16468.706} C_VEL
LIN {X 0,Y 372.814,Z 351.138,A -85,B 0,C 180,E1 -16470,E2 -16470} C_VEL
LIN {X 0,Y 372.515,Z 351.089,A -85,B 0,C 180,E1 -16471.297,E2 -16471.297} C_VEL
LIN {X 0,Y 371.176,Z 350.776,A -85,B 0,C 180,E1 -16473.256,E2 -16473.256} C_VEL
LIN {X 0,Y 369.977,Z 350.428,A -85,B 0,C 180,E1 -16474.358,E2 -16474.358} C_VEL
LIN {X 0,Y 367.56,Z 349.09,A -85,B 0,C 180,E1 -16476.225,E2 -16476.225} C_VEL
LIN {X 0,Y 365.258,Z 347.229,A -85,B 0,C 180,E1 -16477.74,E2 -16477.74} C_VEL
LIN {X 0,Y 362.954,Z 344.831,A -85,B 0,C 180,E1 -16479.121,E2 -16479.121} C_VEL
LIN {X 0,Y 361.057,Z 342.963,A -85,B 0,C 180,E1 -16480.089,E2 -16480.089} C_VEL
LIN {X 0,Y 356.25,Z 339.507,A -85,B 0,C 180,E1 -16481.909,E2 -16481.909} C_VEL
LIN {X 0,Y 351.884,Z 335.317,A -85,B 0,C 180,E1 -16483.501,E2 -16483.501} C_VEL
LIN {X 0,Y 347.219,Z 331.274,A -85,B 0,C 180,E1 -16484.947,E2 -16484.947} C_VEL
LIN {X 0,Y 342.08,Z 326.154,A -85,B 0,C 180,E1 -16486.438,E2 -16486.438} C_VEL
LIN {X 0,Y 336.281,Z 320.284,A -85,B 0,C 180,E1 -16487.916,E2 -16487.916} C_VEL
LIN {X 0,Y 330.592,Z 314.311,A -85,B 0,C 180,E1 -16489.244,E2 -16489.244} C_VEL
LIN {X 0,Y 324.731,Z 307.797,A -85,B 0,C 180,E1 -16490.487,E2 -16490.487} C_VEL
LIN {X 0,Y 319.552,Z 301.782,A -85,B 0,C 180,E1 -16491.497,E2 -16491.497} C_VEL
LIN {X 0,Y 312.034,Z 292.438,A -85,B 0,C 180,E1 -16492.801,E2 -16492.801} C_VEL
LIN {X 0,Y 306.443,Z 284.371,A -85,B 0,C 180,E1 -16493.659,E2 -16493.659} C_VEL
LIN {X 0,Y 301.831,Z 276.63,A -85,B 0,C 180,E1 -16494.323,E2 -16494.323} C_VEL
LIN {X 0,Y 298.639,Z 269.773,A -85,B 0,C 180,E1 -16494.789,E2 -16494.789} C_VEL
LIN {X 0,Y 298.443,Z 268.81,A -85,B 0,C 180,E1 -16494.882,E2 -16494.882} C_VEL
LIN {X 0,Y 298.411,Z 268.816,A -85,B 0,C 180,E1 -16498.1,E2 -16498.1} C_VEL
LIN {X 0,Y 298.348,Z 268.824,A -85,B 0,C 180,E1 -16502.023,E2 -16502.023} C_VEL
LIN {X 0,Y 298.373,Z 268.82,A -85,B 0,C 180,E1 -16506.075,E2 -16506.075} C_VEL
LIN {X 0,Y 298.381,Z 268.818,A -85,B 0,C 180,E1 -16509.49,E2 -16509.49} C_VEL
LIN {X 0,Y 298.427,Z 268.81,A -85,B 0,C 180,E1 -16513.124,E2 -16513.124} C_VEL
LIN {X 0,Y 298.43,Z 268.81,A -85,B 0,C 180,E1 -16516.94,E2 -16516.94} C_VEL
LIN {X 0,Y 298.392,Z 268.815,A -85,B 0,C 180,E1 -16521.008,E2 -16521.008} C_VEL
LIN {X 0,Y 298.396,Z 268.814,A -85,B 0,C 180,E1 -16523.939,E2 -16523.939} C_VEL
LIN {X 0,Y 298.362,Z 268.818,A -85,B 0,C 180,E1 -16527.992,E2 -16527.992} C_VEL
LIN {X 0,Y 298.429,Z 268.809,A -85,B 0,C 180,E1 -16531.912,E2 -16531.912} C_VEL
LIN {X 0,Y 298.456,Z 268.807,A -85,B 0,C 180,E1 -16534.932,E2 -16534.932} C_VEL
LIN {X 0,Y 298.408,Z 268.811,A -85,B 0,C 180,E1 -16539.322,E2 -16539.322} C_VEL
LIN {X 0,Y 298.458,Z 268.806,A -85,B 0,C 180,E1 -16542.184,E2 -16542.184} C_VEL
LIN {X 0,Y 298.569,Z 268.793,A -85,B 0,C 180,E1 -16545.003,E2 -16545.003} C_VEL
LIN {X 0,Y 298.569,Z 268.791,A -85,B 0,C 180,E1 -16549.154,E2 -16549.154} C_VEL
LIN {X 0,Y 298.704,Z 268.775,A -85,B 0,C 180,E1 -16551.893,E2 -16551.893} C_VEL
LIN {X 0,Y 298.63,Z 268.785,A -85,B 0,C 180,E1 -16554.607,E2 -16554.607} C_VEL
LIN {X 0,Y 298.897,Z 268.745,A -85,B 0,C 180,E1 -16558.661,E2 -16558.661} C_VEL
LIN {X 0,Y 298.835,Z 268.756,A -85,B 0,C 180,E1 -16562.01,E2 -16562.01} C_VEL
LIN {X 0,Y 298.731,Z 268.772,A -85,B 0,C 180,E1 -16566.763,E2 -16566.763} C_VEL
LIN {X 0,Y 298.69,Z 268.779,A -85,B 0,C 180,E1 -16567.863,E2 -16567.863} C_VEL
LIN {X 0,Y 298.013,Z 268.868,A -85,B 0,C 180,E1 -16568.988,E2 -16568.988} C_VEL
LIN {X 0,Y 295.065,Z 269.231,A -85,B 0,C 180,E1 -16570.815,E2 -16570.815} C_VEL
LIN {X 0,Y 292.578,Z 269.541,A -85,B 0,C 180,E1 -16572.299,E2 -16572.299} C_VEL
LIN {X 0,Y 291.544,Z 269.669,A -85,B 0,C 180,E1 -16573.45,E2 -16573.45} C_VEL
LIN {X 0,Y 291.478,Z 269.678,A -85,B 0,C 180,E1 -16573.84,E2 -16573.84} C_VEL
LIN {X 0,Y 291.409,Z 269.684,A -85,B 0,C 180,E1 -16576.83,E2 -16576.83} C_VEL
LIN {X 0,Y 291.398,Z 269.689,A -85,B 0,C 180,E1 -16579.849,E2 -16579.849} C_VEL
LIN {X 0,Y 291.333,Z 269.694,A -85,B 0,C 180,E1 -16584.218,E2 -16584.218} C_VEL
LIN {X 0,Y 291.338,Z 269.697,A -85,B 0,C 180,E1 -16587.287,E2 -16587.287} C_VEL
LIN {X 0,Y 291.312,Z 269.699,A -85,B 0,C 180,E1 -16590.447,E2 -16590.447} C_VEL
LIN {X 0,Y 291.352,Z 269.697,A -85,B 0,C 180,E1 -16592.408,E2 -16592.408} C_VEL
LIN {X 0,Y 291.608,Z 271.252,A -85,B 0,C 180,E1 -16595.347,E2 -16595.347} C_VEL
LIN {X 0,Y 291.95,Z 274.003,A -85,B 0,C 180,E1 -16599.618,E2 -16599.618} C_VEL
LIN {X 0,Y 292.221,Z 275.903,A -85,B 0,C 180,E1 -16602.338,E2 -16602.338} C_VEL
LIN {X 0,Y 292.572,Z 278.771,A -85,B 0,C 180,E1 -16606.115,E2 -16606.115} C_VEL
LIN {X 0,Y 292.543,Z 280.437,A -85,B 0,C 180,E1 -16608.145,E2 -16608.145} C_VEL
LIN {X 0,Y 292.176,Z 283.181,A -85,B 0,C 180,E1 -16611.289,E2 -16611.289} C_VEL
LIN {X 0,Y 291.627,Z 286.653,A -85,B 0,C 180,E1 -16615.031,E2 -16615.031} C_VEL
LIN {X 0,Y 291.159,Z 289.462,A -85,B 0,C 180,E1 -16617.925,E2 -16617.925} C_VEL
LIN {X 0,Y 290.729,Z 292.639,A -85,B 0,C 180,E1 -16621.088,E2 -16621.088} C_VEL
LIN {X 0,Y 290.24,Z 296.436,A -85,B 0,C 180,E1 -16624.773,E2 -16624.773} C_VEL
LIN {X 0,Y 292.253,Z 304.329,A -85,B 0,C 180,E1 -16625.3,E2 -16625.3} C_VEL
LIN {X 0,Y 294.781,Z 315.05,A -85,B 0,C 180,E1 -16626.162,E2 -16626.162} C_VEL
LIN {X 0,Y 296.318,Z 323.538,A -85,B 0,C 180,E1 -16626.941,E2 -16626.941} C_VEL
LIN {X 0,Y 297.577,Z 333.988,A -85,B 0,C 180,E1 -16628.05,E2 -16628.05} C_VEL
LIN {X 0,Y 298.292,Z 342.717,A -85,B 0,C 180,E1 -16629.126,E2 -16629.126} C_VEL
LIN {X 0,Y 296.982,Z 351.651,A -85,B 0,C 180,E1 -16630.293,E2 -16630.293} C_VEL
LIN {X 0,Y 295.572,Z 360.182,A -85,B 0,C 180,E1 -16631.636,E2 -16631.636} C_VEL
LIN {X 0,Y 294.425,Z 367.717,A -85,B 0,C 180,E1 -16633.066,E2 -16633.066} C_VEL
LIN {X 0,Y 293.366,Z 373.611,A -85,B 0,C 180,E1 -16634.365,E2 -16634.365} C_VEL
LIN {X 0,Y 292.203,Z 380.151,A -85,B 0,C 180,E1 -16636.083,E2 -16636.083} C_VEL
LIN {X 0,Y 291.377,Z 384.653,A -85,B 0,C 180,E1 -16637.463,E2 -16637.463} C_VEL
LIN {X 0,Y 290.527,Z 390.15,A -85,B 0,C 180,E1 -16639.547,E2 -16639.547} C_VEL
LIN {X 0,Y 289.93,Z 394.479,A -85,B 0,C 180,E1 -16641.637,E2 -16641.637} C_VEL
LIN {X 0,Y 289.685,Z 396.849,A -85,B 0,C 180,E1 -16643.033,E2 -16643.033} C_VEL
LIN {X 0,Y 289.519,Z 398.703,A -85,B 0,C 180,E1 -16644.468,E2 -16644.468} C_VEL
LIN {X 0,Y 289.451,Z 401.104,A -85,B 0,C 180,E1 -16647.217,E2 -16647.217} C_VEL
LIN {X 0,Y 289.414,Z 401.693,A -85,B 0,C 180,E1 -16648.609,E2 -16648.609} C_VEL
LIN {X 0,Y 289.414,Z 401.693,A -85,B 0,C 180,E1 -16651.391,E2 -16651.391} C_VEL
LIN {X 0,Y 289.451,Z 401.104,A -85,B 0,C 180,E1 -16652.783,E2 -16652.783} C_VEL
LIN {X 0,Y 289.539,Z 398.652,A -85,B 0,C 180,E1 -16655.572,E2 -16655.572} C_VEL
LIN {X 0,Y 289.767,Z 395.697,A -85,B 0,C 180,E1 -16657.666,E2 -16657.666} C_VEL
LIN {X 0,Y 290.309,Z 391.705,A -85,B 0,C 180,E1 -16659.756,E2 -16659.756} C_VEL
LIN {X 0,Y 291.066,Z 386.571,A -85,B 0,C 180,E1 -16661.843,E2 -16661.843} C_VEL
LIN {X 0,Y 291.978,Z 381.306,A -85,B 0,C 180,E1 -16663.573,E2 -16663.573} C_VEL
LIN {X 0,Y 293.103,Z 374.987,A -85,B 0,C 180,E1 -16665.293,E2 -16665.293} C_VEL
LIN {X 0,Y 294.193,Z 369.035,A -85,B 0,C 180,E1 -16666.658,E2 -16666.658} C_VEL
LIN {X 0,Y 295.268,Z 362.103,A -85,B 0,C 180,E1 -16668.024,E2 -16668.024} C_VEL
LIN {X 0,Y 296.568,Z 353.92,A -85,B 0,C 180,E1 -16669.376,E2 -16669.376} C_VEL
LIN {X 0,Y 297.969,Z 345.41,A -85,B 0,C 180,E1 -16670.539,E2 -16670.539} C_VEL
LIN {X 0,Y 298.165,Z 341.372,A -85,B 0,C 180,E1 -16671.062,E2 -16671.062} C_VEL
LIN {X 0,Y 297.179,Z 330.019,A -85,B 0,C 180,E1 -16672.402,E2 -16672.402} C_VEL
LIN {X 0,Y 295.556,Z 318.831,A -85,B 0,C 180,E1 -16673.501,E2 -16673.501} C_VEL
LIN {X 0,Y 293.157,Z 307.906,A -85,B 0,C 180,E1 -16674.428,E2 -16674.428} C_VEL
LIN {X 0,Y 290.374,Z 297.573,A -85,B 0,C 180,E1 -16675.168,E2 -16675.168} C_VEL
LIN {X 0,Y 290.241,Z 296.437,A -85,B 0,C 180,E1 -16675.226,E2 -16675.226} C_VEL
LIN {X 0,Y 290.804,Z 291.997,A -85,B 0,C 180,E1 -16679.528,E2 -16679.528} C_VEL
LIN {X 0,Y 291.402,Z 287.877,A -85,B 0,C 180,E1 -16683.69,E2 -16683.69} C_VEL
LIN {X 0,Y 291.997,Z 284.366,A -85,B 0,C 180,E1 -16687.405,E2 -16687.405} C_VEL
LIN {X 0,Y 292.389,Z 281.619,A -85,B 0,C 180,E1 -16690.464,E2 -16690.464} C_VEL
LIN {X 0,Y 292.571,Z 280.077,A -85,B 0,C 180,E1 -16692.267,E2 -16692.267} C_VEL
LIN {X 0,Y 292.562,Z 278.533,A -85,B 0,C 180,E1 -16694.157,E2 -16694.157} C_VEL
LIN {X 0,Y 292.223,Z 275.889,A -85,B 0,C 180,E1 -16697.662,E2 -16697.662} C_VEL
LIN {X 0,Y 291.864,Z 273.417,A -85,B 0,C 180,E1 -16701.232,E2 -16701.232} C_VEL
LIN {X 0,Y 291.56,Z 271.026,A -85,B 0,C 180,E1 -16705.04,E2 -16705.04} C_VEL
LIN {X 0,Y 291.377,Z 269.691,A -85,B 0,C 180,E1 -16707.944,E2 -16707.944} C_VEL
LIN {X 0,Y 291.324,Z 269.697,A -85,B 0,C 180,E1 -16711.145,E2 -16711.145} C_VEL
LIN {X 0,Y 291.35,Z 269.697,A -85,B 0,C 180,E1 -16714.258,E2 -16714.258} C_VEL
LIN {X 0,Y 291.357,Z 269.693,A -85,B 0,C 180,E1 -16717.29,E2 -16717.29} C_VEL
LIN {X 0,Y 291.391,Z 269.692,A -85,B 0,C 180,E1 -16720.258,E2 -16720.258} C_VEL
LIN {X 0,Y 291.478,Z 269.676,A -85,B 0,C 180,E1 -16724.676,E2 -16724.676} C_VEL
LIN {X 0,Y 291.529,Z 269.669,A -85,B 0,C 180,E1 -16728.873,E2 -16728.873} C_VEL
LIN {X 0,Y 291.651,Z 269.657,A -85,B 0,C 180,E1 -16731.679,E2 -16731.679} C_VEL
LIN {X 0,Y 291.593,Z 269.661,A -85,B 0,C 180,E1 -16734.46,E2 -16734.46} C_VEL
LIN {X 0,Y 291.873,Z 269.624,A -85,B 0,C 180,E1 -16738.612,E2 -16738.612} C_VEL
LIN {X 0,Y 291.865,Z 269.619,A -85,B 0,C 180,E1 -16741.372,E2 -16741.372} C_VEL
LIN {X 0,Y 291.693,Z 269.649,A -85,B 0,C 180,E1 -16746.911,E2 -16746.911} C_VEL
LIN {X 0,Y 291.555,Z 269.666,A -85,B 0,C 180,E1 -16749.706,E2 -16749.706} C_VEL
LIN {X 0,Y 291.498,Z 269.671,A -85,B 0,C 180,E1 -16753.942,E2 -16753.942} C_VEL
LIN {X 0,Y 291.414,Z 269.684,A -85,B 0,C 180,E1 -16756.813,E2 -16756.813} C_VEL
LIN {X 0,Y 291.403,Z 269.681,A -85,B 0,C 180,E1 -16759.852,E2 -16759.852} C_VEL
LIN {X 0,Y 291.357,Z 269.689,A -85,B 0,C 180,E1 -16764.199,E2 -16764.199} C_VEL
LIN {X 0,Y 291.392,Z 269.688,A -85,B 0,C 180,E1 -16767.264,E2 -16767.264} C_VEL
LIN {X 0,Y 291.304,Z 269.699,A -85,B 0,C 180,E1 -16770.429,E2 -16770.429} C_VEL
LIN {X 0,Y 291.312,Z 269.695,A -85,B 0,C 180,E1 -16773.691,E2 -16773.691} C_VEL
LIN {X 0,Y 291.362,Z 269.69,A -85,B 0,C 180,E1 -16777.252,E2 -16777.252} C_VEL
LIN {X 0,Y 291.363,Z 269.693,A -85,B 0,C 180,E1 -16780.624,E2 -16780.624} C_VEL
LIN {X 0,Y 291.366,Z 269.693,A -85,B 0,C 180,E1 -16784.373,E2 -16784.373} C_VEL
LIN {X 0,Y 291.345,Z 269.695,A -85,B 0,C 180,E1 -16788.384,E2 -16788.384} C_VEL
LIN {X 0,Y 291.332,Z 269.694,A -85,B 0,C 180,E1 -16791.156,E2 -16791.156} C_VEL
LIN {X 0,Y 291.315,Z 269.697,A -85,B 0,C 180,E1 -16794.62,E2 -16794.62} C_VEL
LIN {X 0,Y 291.325,Z 269.699,A -85,B 0,C 180,E1 -16797.946,E2 -16797.946} C_VEL
LIN {X 0,Y 291.331,Z 269.695,A -85,B 0,C 180,E1 -16801.153,E2 -16801.153} C_VEL
LIN {X 0,Y 291.403,Z 269.686,A -85,B 0,C 180,E1 -16804.525,E2 -16804.525} C_VEL
LIN {X 0,Y 292.44,Z 272.615,A -85,B 0,C 180,E1 -16804.72,E2 -16804.72} C_VEL
LIN {X 0,Y 297.903,Z 283.604,A -85,B 0,C 180,E1 -16805.575,E2 -16805.575} C_VEL
LIN {X 0,Y 303.777,Z 292.88,A -85,B 0,C 180,E1 -16806.53,E2 -16806.53} C_VEL
LIN {X 0,Y 311.184,Z 302.758,A -85,B 0,C 180,E1 -16807.787,E2 -16807.787} C_VEL
LIN {X 0,Y 318.195,Z 311.012,A -85,B 0,C 180,E1 -16809.088,E2 -16809.088} C_VEL
LIN {X 0,Y 324.943,Z 318.602,A -85,B 0,C 180,E1 -16810.504,E2 -16810.504} C_VEL
LIN {X 0,Y 330.853,Z 324.914,A -85,B 0,C 180,E1 -16811.883,E2 -16811.883} C_VEL
LIN {X 0,Y 337.13,Z 331.292,A -85,B 0,C 180,E1 -16813.488,E2 -16813.488} C_VEL
LIN {X 0,Y 342.086,Z 336.104,A -85,B 0,C 180,E1 -16814.887,E2 -16814.887} C_VEL
LIN {X 0,Y 348.118,Z 341.499,A -85,B 0,C 180,E1 -16816.812,E2 -16816.812} C_VEL
LIN {X 0,Y 351.797,Z 344.989,A -85,B 0,C 180,E1 -16818.158,E2 -16818.158} C_VEL
LIN {X 0,Y 356.02,Z 348.075,A -85,B 0,C 180,E1 -16819.766,E2 -16819.766} C_VEL
LIN {X 0,Y 359.381,Z 351.355,A -85,B 0,C 180,E1 -16821.547,E2 -16821.547} C_VEL
LIN {X 0,Y 362.154,Z 353.865,A -85,B 0,C 180,E1 -16823.314,E2 -16823.314} C_VEL
LIN {X 0,Y 363.768,Z 354.966,A -85,B 0,C 180,E1 -16824.457,E2 -16824.457} C_VEL
LIN {X 0,Y 366.122,Z 356.052,A -85,B 0,C 180,E1 -16826.384,E2 -16826.384} C_VEL
LIN {X 0,Y 367.396,Z 356.419,A -85,B 0,C 180,E1 -16827.807,E2 -16827.807} C_VEL
LIN {X 0,Y 368.022,Z 356.511,A -85,B 0,C 180,E1 -16828.906,E2 -16828.906} C_VEL
LIN {X 0,Y 368.228,Z 356.538,A -85,B 0,C 180,E1 -16830,E2 -16830} C_VEL
LIN {X 0,Y 368.017,Z 356.5,A -85,B 0,C 180,E1 -16831.094,E2 -16831.094} C_VEL
LIN {X 0,Y 367.393,Z 356.401,A -85,B 0,C 180,E1 -16832.193,E2 -16832.193} C_VEL
LIN {X 0,Y 366.122,Z 356.055,A -85,B 0,C 180,E1 -16833.617,E2 -16833.617} C_VEL
LIN {X 0,Y 363.773,Z 354.997,A -85,B 0,C 180,E1 -16835.543,E2 -16835.543} C_VEL
LIN {X 0,Y 361.27,Z 353.164,A -85,B 0,C 180,E1 -16837.271,E2 -16837.271} C_VEL
LIN {X 0,Y 358.418,Z 350.324,A -85,B 0,C 180,E1 -16839.025,E2 -16839.025} C_VEL
LIN {X 0,Y 355.999,Z 348.081,A -85,B 0,C 180,E1 -16840.234,E2 -16840.234} C_VEL
LIN {X 0,Y 351.106,Z 344.392,A -85,B 0,C 180,E1 -16842.086,E2 -16842.086} C_VEL
LIN {X 0,Y 346.982,Z 340.456,A -85,B 0,C 180,E1 -16843.58,E2 -16843.58} C_VEL
LIN {X 0,Y 342.072,Z 336.11,A -85,B 0,C 180,E1 -16845.104,E2 -16845.104} C_VEL
LIN {X 0,Y 337.142,Z 331.258,A -85,B 0,C 180,E1 -16846.519,E2 -16846.519} C_VEL
LIN {X 0,Y 330.865,Z 324.897,A -85,B 0,C 180,E1 -16848.121,E2 -16848.121} C_VEL
LIN {X 0,Y 324.88,Z 318.557,A -85,B 0,C 180,E1 -16849.502,E2 -16849.502} C_VEL
LIN {X 0,Y 318.181,Z 311.035,A -85,B 0,C 180,E1 -16850.911,E2 -16850.911} C_VEL
LIN {X 0,Y 311.178,Z 302.706,A -85,B 0,C 180,E1 -16852.21,E2 -16852.21} C_VEL
LIN {X 0,Y 304.644,Z 294.056,A -85,B 0,C 180,E1 -16853.326,E2 -16853.326} C_VEL
LIN {X 0,Y 298.823,Z 285.273,A -85,B 0,C 180,E1 -16854.274,E2 -16854.274} C_VEL
LIN {X 0,Y 294.424,Z 276.748,A -85,B 0,C 180,E1 -16854.98,E2 -16854.98} C_VEL
LIN {X 0,Y 291.585,Z 270.708,A -85,B 0,C 180,E1 -16855.412,E2 -16855.412} C_VEL
LIN {X 0,Y 291.392,Z 269.688,A -85,B 0,C 180,E1 -16855.505,E2 -16855.505} C_VEL
LIN {X 0,Y 291.337,Z 269.696,A -85,B 0,C 180,E1 -16859.745,E2 -16859.745} C_VEL
LIN {X 0,Y 291.296,Z 269.701,A -85,B 0,C 180,E1 -16863.704,E2 -16863.704} C_VEL
LIN {X 0,Y 291.342,Z 269.693,A -85,B 0,C 180,E1 -16867.263,E2 -16867.263} C_VEL
LIN {X 0,Y 291.357,Z 269.69,A -85,B 0,C 180,E1 -16870.637,E2 -16870.637} C_VEL
LIN {X 0,Y 291.365,Z 269.689,A -85,B 0,C 180,E1 -16874.387,E2 -16874.387} C_VEL
LIN {X 0,Y 291.35,Z 269.691,A -85,B 0,C 180,E1 -16878.398,E2 -16878.398} C_VEL
LIN {X 0,Y 291.341,Z 269.695,A -85,B 0,C 180,E1 -16881.17,E2 -16881.17} C_VEL
LIN {X 0,Y 291.351,Z 269.691,A -85,B 0,C 180,E1 -16884.637,E2 -16884.637} C_VEL
LIN {X 0,Y 291.339,Z 269.693,A -85,B 0,C 180,E1 -16887.958,E2 -16887.958} C_VEL
LIN {X 0,Y 291.349,Z 269.695,A -85,B 0,C 180,E1 -16891.166,E2 -16891.166} C_VEL
LIN {X 0,Y 291.385,Z 269.685,A -85,B 0,C 180,E1 -16894.28,E2 -16894.28} C_VEL
LIN {X 0,Y 291.349,Z 269.693,A -85,B 0,C 180,E1 -16897.307,E2 -16897.307} C_VEL
LIN {X 0,Y 291.419,Z 269.68,A -85,B 0,C 180,E1 -16900.277,E2 -16900.277} C_VEL
LIN {X 0,Y 291.481,Z 269.676,A -85,B 0,C 180,E1 -16904.674,E2 -16904.674} C_VEL
LIN {X 0,Y 291.514,Z 269.671,A -85,B 0,C 180,E1 -16908.889,E2 -16908.889} C_VEL
LIN {X 0,Y 291.654,Z 269.652,A -85,B 0,C 180,E1 -16911.696,E2 -16911.696} C_VEL
LIN {X 0,Y 291.6,Z 269.661,A -85,B 0,C 180,E1 -16914.476,E2 -16914.476} C_VEL
LIN {X 0,Y 291.865,Z 269.619,A -85,B 0,C 180,E1 -16918.628,E2 -16918.628} C_VEL
LIN {X 0,Y 291.873,Z 269.624,A -85,B 0,C 180,E1 -16921.388,E2 -16921.388} C_VEL
LIN {X 0,Y 291.684,Z 269.65,A -85,B 0,C 180,E1 -16926.927,E2 -16926.927} C_VEL
LIN {X 0,Y 291.569,Z 269.666,A -85,B 0,C 180,E1 -16929.721,E2 -16929.721} C_VEL
LIN {X 0,Y 291.478,Z 269.678,A -85,B 0,C 180,E1 -16933.84,E2 -16933.84} C_VEL
LIN {X 0,Y 290.834,Z 269.764,A -85,B 0,C 180,E1 -16934.993,E2 -16934.993} C_VEL
LIN {X 0,Y 287.908,Z 270.125,A -85,B 0,C 180,E1 -16936.867,E2 -16936.867} C_VEL
LIN {X 0,Y 285.425,Z 270.43,A -85,B 0,C 180,E1 -16938.389,E2 -16938.389} C_VEL
LIN {X 0,Y 284.396,Z 270.561,A -85,B 0,C 180,E1 -16939.571,E2 -16939.571} C_VEL
LIN {X 0,Y 284.334,Z 270.567,A -85,B 0,C 180,E1 -16939.971,E2 -16939.971} C_VEL
LIN {X 0,Y 284.301,Z 270.572,A -85,B 0,C 180,E1 -16943.846,E2 -16943.846} C_VEL
LIN {X 0,Y 284.295,Z 270.573,A -85,B 0,C 180,E1 -16947.135,E2 -16947.135} C_VEL
LIN {X 0,Y 284.284,Z 270.576,A -85,B 0,C 180,E1 -16950.089,E2 -16950.089} C_VEL
LIN {X 0,Y 284.371,Z 271.002,A -85,B 0,C 180,E1 -16952.944,E2 -16952.944} C_VEL
LIN {X 0,Y 284.625,Z 272.965,A -85,B 0,C 180,E1 -16956.35,E2 -16956.35} C_VEL
LIN {X 0,Y 284.977,Z 275.385,A -85,B 0,C 180,E1 -16960.138,E2 -16960.138} C_VEL
LIN {X 0,Y 285.334,Z 277.817,A -85,B 0,C 180,E1 -16963.611,E2 -16963.611} C_VEL
LIN {X 0,Y 285.537,Z 279.966,A -85,B 0,C 180,E1 -16966.436,E2 -16966.436} C_VEL
LIN {X 0,Y 285.326,Z 282.721,A -85,B 0,C 180,E1 -16969.789,E2 -16969.789} C_VEL
LIN {X 0,Y 284.728,Z 286.152,A -85,B 0,C 180,E1 -16973.673,E2 -16973.673} C_VEL
LIN {X 0,Y 284.168,Z 289.488,A -85,B 0,C 180,E1 -16977.243,E2 -16977.243} C_VEL
LIN {X 0,Y 283.738,Z 292.454,A -85,B 0,C 180,E1 -16980.305,E2 -16980.305} C_VEL
LIN {X 0,Y 283.242,Z 296.449,A -85,B 0,C 180,E1 -16984.119,E2 -16984.119} C_VEL
LIN {X 0,Y 285.888,Z 306.507,A -85,B 0,C 180,E1 -16984.844,E2 -16984.844} C_VEL
LIN {X 0,Y 288.153,Z 316.282,A -85,B 0,C 180,E1 -16985.686,E2 -16985.686} C_VEL
LIN {X 0,Y 289.686,Z 325.052,A -85,B 0,C 180,E1 -16986.544,E2 -16986.544} C_VEL
LIN {X 0,Y 290.728,Z 333.74,A -85,B 0,C 180,E1 -16987.502,E2 -16987.502} C_VEL
LIN {X 0,Y 291.399,Z 342.603,A -85,B 0,C 180,E1 -16988.622,E2 -16988.622} C_VEL
LIN {X 0,Y 291.095,Z 346.55,A -85,B 0,C 180,E1 -16989.139,E2 -16989.139} C_VEL
LIN {X 0,Y 289.128,Z 358.049,A -85,B 0,C 180,E1 -16990.844,E2 -16990.844} C_VEL
LIN {X 0,Y 287.694,Z 366.869,A -85,B 0,C 180,E1 -16992.514,E2 -16992.514} C_VEL
LIN {X 0,Y 286.483,Z 373.398,A -85,B 0,C 180,E1 -16993.98,E2 -16993.98} C_VEL
LIN {X 0,Y 285.282,Z 379.938,A -85,B 0,C 180,E1 -16995.739,E2 -16995.739} C_VEL
LIN {X 0,Y 284.418,Z 384.441,A -85,B 0,C 180,E1 -16997.151,E2 -16997.151} C_VEL
LIN {X 0,Y 283.531,Z 389.938,A -85,B 0,C 180,E1 -16999.286,E2 -16999.286} C_VEL
LIN {X 0,Y 282.896,Z 394.267,A -85,B 0,C 180,E1 -17001.428,E2 -17001.428} C_VEL
LIN {X 0,Y 282.614,Z 396.637,A -85,B 0,C 180,E1 -17002.858,E2 -17002.858} C_VEL
LIN {X 0,Y 282.427,Z 398.751,A -85,B 0,C 180,E1 -17004.536,E2 -17004.536} C_VEL
LIN {X 0,Y 282.36,Z 400.892,A -85,B 0,C 180,E1 -17007.147,E2 -17007.147} C_VEL
LIN {X 0,Y 282.339,Z 401.483,A -85,B 0,C 180,E1 -17008.574,E2 -17008.574} C_VEL
LIN {X 0,Y 282.339,Z 401.483,A -85,B 0,C 180,E1 -17011.426,E2 -17011.426} C_VEL
LIN {X 0,Y 282.36,Z 400.892,A -85,B 0,C 180,E1 -17012.853,E2 -17012.853} C_VEL
LIN {X 0,Y 282.464,Z 398.44,A -85,B 0,C 180,E1 -17015.712,E2 -17015.712} C_VEL
LIN {X 0,Y 282.723,Z 395.485,A -85,B 0,C 180,E1 -17017.858,E2 -17017.858} C_VEL
LIN {X 0,Y 283.273,Z 391.493,A -85,B 0,C 180,E1 -17020.001,E2 -17020.001} C_VEL
LIN {X 0,Y 284.089,Z 386.358,A -85,B 0,C 180,E1 -17022.138,E2 -17022.138} C_VEL
LIN {X 0,Y 285.064,Z 381.094,A -85,B 0,C 180,E1 -17023.909,E2 -17023.909} C_VEL
LIN {X 0,Y 286.214,Z 374.774,A -85,B 0,C 180,E1 -17025.67,E2 -17025.67} C_VEL
LIN {X 0,Y 287.565,Z 367.789,A -85,B 0,C 180,E1 -17027.287,E2 -17027.287} C_VEL
LIN {X 0,Y 288.802,Z 359.97,A -85,B 0,C 180,E1 -17028.81,E2 -17028.81} C_VEL
LIN {X 0,Y 290.289,Z 351.439,A -85,B 0,C 180,E1 -17030.181,E2 -17030.181} C_VEL
LIN {X 0,Y 291.426,Z 343.843,A -85,B 0,C 180,E1 -17031.207,E2 -17031.207} C_VEL
LIN {X 0,Y 290.881,Z 335.652,A -85,B 0,C 180,E1 -17032.268,E2 -17032.268} C_VEL
LIN {X 0,Y 289.857,Z 326.386,A -85,B 0,C 180,E1 -17033.317,E2 -17033.317} C_VEL
LIN {X 0,Y 288.43,Z 317.556,A -85,B 0,C 180,E1 -17034.195,E2 -17034.195} C_VEL
LIN {X 0,Y 286.034,Z 306.97,A -85,B 0,C 180,E1 -17035.116,E2 -17035.116} C_VEL
LIN {X 0,Y 283.331,Z 297.261,A -85,B 0,C 180,E1 -17035.842,E2 -17035.842} C_VEL
LIN {X 0,Y 283.218,Z 296.223,A -85,B 0,C 180,E1 -17035.913,E2 -17035.913} C_VEL
LIN {X 0,Y 283.768,Z 292.245,A -85,B 0,C 180,E1 -17039.897,E2 -17039.897} C_VEL
LIN {X 0,Y 284.201,Z 289.285,A -85,B 0,C 180,E1 -17042.958,E2 -17042.958} C_VEL
LIN {X 0,Y 284.743,Z 286.152,A -85,B 0,C 180,E1 -17046.324,E2 -17046.324} C_VEL
LIN {X 0,Y 285.312,Z 282.716,A -85,B 0,C 180,E1 -17050.208,E2 -17050.208} C_VEL
LIN {X 0,Y 285.543,Z 279.946,A -85,B 0,C 180,E1 -17053.562,E2 -17053.562} C_VEL
LIN {X 0,Y 285.345,Z 277.81,A -85,B 0,C 180,E1 -17056.391,E2 -17056.391} C_VEL
LIN {X 0,Y 284.95,Z 275.217,A -85,B 0,C 180,E1 -17060.106,E2 -17060.106} C_VEL
LIN {X 0,Y 284.572,Z 272.405,A -85,B 0,C 180,E1 -17064.585,E2 -17064.585} C_VEL
LIN {X 0,Y 284.364,Z 270.933,A -85,B 0,C 180,E1 -17067.17,E2 -17067.17} C_VEL
LIN {X 0,Y 284.319,Z 270.571,A -85,B 0,C 180,E1 -17070.364,E2 -17070.364} C_VEL
LIN {X 0,Y 284.304,Z 270.571,A -85,B 0,C 180,E1 -17073.572,E2 -17073.572} C_VEL
LIN {X 0,Y 284.315,Z 270.573,A -85,B 0,C 180,E1 -17076.695,E2 -17076.695} C_VEL
LIN {X 0,Y 284.341,Z 270.569,A -85,B 0,C 180,E1 -17079.921,E2 -17079.921} C_VEL
LIN {X 0,Y 284.419,Z 270.557,A -85,B 0,C 180,E1 -17084.509,E2 -17084.509} C_VEL
LIN {X 0,Y 284.46,Z 270.55,A -85,B 0,C 180,E1 -17088.593,E2 -17088.593} C_VEL
LIN {X 0,Y 284.608,Z 270.532,A -85,B 0,C 180,E1 -17091.472,E2 -17091.472} C_VEL
LIN {X 0,Y 284.564,Z 270.538,A -85,B 0,C 180,E1 -17094.323,E2 -17094.323} C_VEL
LIN {X 0,Y 284.839,Z 270.5,A -85,B 0,C 180,E1 -17098.578,E2 -17098.578} C_VEL
LIN {X 0,Y 284.832,Z 270.494,A -85,B 0,C 180,E1 -17101.406,E2 -17101.406} C_VEL
LIN {X 0,Y 284.647,Z 270.528,A -85,B 0,C 180,E1 -17107.083,E2 -17107.083} C_VEL
LIN {X 0,Y 284.501,Z 270.543,A -85,B 0,C 180,E1 -17109.949,E2 -17109.949} C_VEL
LIN {X 0,Y 284.446,Z 270.549,A -85,B 0,C 180,E1 -17114.295,E2 -17114.295} C_VEL
LIN {X 0,Y 284.343,Z 270.566,A -85,B 0,C 180,E1 -17118.733,E2 -17118.733} C_VEL
LIN {X 0,Y 284.293,Z 270.57,A -85,B 0,C 180,E1 -17121.756,E2 -17121.756} C_VEL
LIN {X 0,Y 284.311,Z 270.569,A -85,B 0,C 180,E1 -17124.838,E2 -17124.838} C_VEL
LIN {X 0,Y 284.3,Z 270.569,A -85,B 0,C 180,E1 -17128.003,E2 -17128.003} C_VEL
LIN {X 0,Y 284.263,Z 270.575,A -85,B 0,C 180,E1 -17131.266,E2 -17131.266} C_VEL
LIN {X 0,Y 284.328,Z 270.566,A -85,B 0,C 180,E1 -17135.346,E2 -17135.346} C_VEL
LIN {X 0,Y 284.295,Z 270.572,A -85,B 0,C 180,E1 -17138.158,E2 -17138.158} C_VEL
LIN {X 0,Y 284.304,Z 270.572,A -85,B 0,C 180,E1 -17142.133,E2 -17142.133} C_VEL
LIN {X 0,Y 284.311,Z 270.572,A -85,B 0,C 180,E1 -17146.201,E2 -17146.201} C_VEL
LIN {X 0,Y 284.308,Z 270.571,A -85,B 0,C 180,E1 -17150.007,E2 -17150.007} C_VEL
LIN {X 0,Y 284.291,Z 270.572,A -85,B 0,C 180,E1 -17153.609,E2 -17153.609} C_VEL
LIN {X 0,Y 284.26,Z 270.575,A -85,B 0,C 180,E1 -17157.184,E2 -17157.184} C_VEL
LIN {X 0,Y 284.308,Z 270.571,A -85,B 0,C 180,E1 -17160.371,E2 -17160.371} C_VEL
LIN {X 0,Y 284.348,Z 270.691,A -85,B 0,C 180,E1 -17163.887,E2 -17163.887} C_VEL
LIN {X 0,Y 285.359,Z 273.452,A -85,B 0,C 180,E1 -17164.063,E2 -17164.063} C_VEL
LIN {X 0,Y 291.767,Z 286.57,A -85,B 0,C 180,E1 -17165.145,E2 -17165.145} C_VEL
LIN {X 0,Y 297.24,Z 295.788,A -85,B 0,C 180,E1 -17166.151,E2 -17166.151} C_VEL
LIN {X 0,Y 305.144,Z 306.513,A -85,B 0,C 180,E1 -17167.596,E2 -17167.596} C_VEL
LIN {X 0,Y 311.958,Z 314.737,A -85,B 0,C 180,E1 -17168.872,E2 -17168.872} C_VEL
LIN {X 0,Y 319.267,Z 322.94,A -85,B 0,C 180,E1 -17170.39,E2 -17170.39} C_VEL
LIN {X 0,Y 325.41,Z 329.513,A -85,B 0,C 180,E1 -17171.824,E2 -17171.824} C_VEL
LIN {X 0,Y 331.881,Z 336.067,A -85,B 0,C 180,E1 -17173.464,E2 -17173.464} C_VEL
LIN {X 0,Y 337.402,Z 341.442,A -85,B 0,C 180,E1 -17175.05,E2 -17175.05} C_VEL
LIN {X 0,Y 341.335,Z 344.898,A -85,B 0,C 180,E1 -17176.262,E2 -17176.262} C_VEL
LIN {X 0,Y 347.028,Z 350.203,A -85,B 0,C 180,E1 -17178.316,E2 -17178.316} C_VEL
LIN {X 0,Y 350.426,Z 352.708,A -85,B 0,C 180,E1 -17179.601,E2 -17179.601} C_VEL
LIN {X 0,Y 352.976,Z 354.945,A -85,B 0,C 180,E1 -17180.835,E2 -17180.835} C_VEL
LIN {X 0,Y 354.977,Z 357.031,A -85,B 0,C 180,E1 -17182.034,E2 -17182.034} C_VEL
LIN {X 0,Y 356.842,Z 358.618,A -85,B 0,C 180,E1 -17183.214,E2 -17183.214} C_VEL
LIN {X 0,Y 359.623,Z 360.427,A -85,B 0,C 180,E1 -17185.207,E2 -17185.207} C_VEL
LIN {X 0,Y 361.332,Z 361.117,A -85,B 0,C 180,E1 -17186.655,E2 -17186.655} C_VEL
LIN {X 0,Y 362.318,Z 361.428,A -85,B 0,C 180,E1 -17187.777,E2 -17187.777} C_VEL
LIN {X 0,Y 362.981,Z 361.535,A -85,B 0,C 180,E1 -17188.891,E2 -17188.891} C_VEL
LIN {X 0,Y 363.205,Z 361.559,A -85,B 0,C 180,E1 -17190,E2 -17190} C_VEL
LIN {X 0,Y 362.976,Z 361.525,A -85,B 0,C 180,E1 -17191.109,E2 -17191.109} C_VEL
LIN {X 0,Y 362.316,Z 361.411,A -85,B 0,C 180,E1 -17192.223,E2 -17192.223} C_VEL
LIN {X 0,Y 361.32,Z 361.113,A -85,B 0,C 180,E1 -17193.345,E2 -17193.345} C_VEL
LIN {X 0,Y 359.623,Z 360.456,A -85,B 0,C 180,E1 -17194.793,E2 -17194.793} C_VEL
LIN {X 0,Y 356.819,Z 358.625,A -85,B 0,C 180,E1 -17196.787,E2 -17196.787} C_VEL
LIN {X 0,Y 354.847,Z 356.854,A -85,B 0,C 180,E1 -17198.065,E2 -17198.065} C_VEL
LIN {X 0,Y 352.081,Z 354.046,A -85,B 0,C 180,E1 -17199.653,E2 -17199.653} C_VEL
LIN {X 0,Y 348.659,Z 351.502,A -85,B 0,C 180,E1 -17201.049,E2 -17201.049} C_VEL
LIN {X 0,Y 345.259,Z 348.613,A -85,B 0,C 180,E1 -17202.34,E2 -17202.34} C_VEL
LIN {X 0,Y 340.407,Z 344.126,A -85,B 0,C 180,E1 -17204.028,E2 -17204.028} C_VEL
LIN {X 0,Y 335.497,Z 339.507,A -85,B 0,C 180,E1 -17205.544,E2 -17205.544} C_VEL
LIN {X 0,Y 328.429,Z 332.669,A -85,B 0,C 180,E1 -17207.432,E2 -17207.432} C_VEL
LIN {X 0,Y 321.29,Z 325.135,A -85,B 0,C 180,E1 -17209.154,E2 -17209.154} C_VEL
LIN {X 0,Y 315.077,Z 318.27,A -85,B 0,C 180,E1 -17210.503,E2 -17210.503} C_VEL
LIN {X 0,Y 308.811,Z 310.92,A -85,B 0,C 180,E1 -17211.735,E2 -17211.735} C_VEL
LIN {X 0,Y 300.272,Z 300.121,A -85,B 0,C 180,E1 -17213.297,E2 -17213.297} C_VEL
LIN {X 0,Y 294.056,Z 290.721,A -85,B 0,C 180,E1 -17214.428,E2 -17214.428} C_VEL
LIN {X 0,Y 289.532,Z 282.088,A -85,B 0,C 180,E1 -17215.257,E2 -17215.257} C_VEL
LIN {X 0,Y 284.512,Z 271.517,A -85,B 0,C 180,E1 -17216.074,E2 -17216.074} C_VEL
LIN {X 0,Y 284.338,Z 270.568,A -85,B 0,C 180,E1 -17216.14,E2 -17216.14} C_VEL
LIN {X 0,Y 284.265,Z 270.578,A -85,B 0,C 180,E1 -17220.103,E2 -17220.103} C_VEL
LIN {X 0,Y 284.258,Z 270.575,A -85,B 0,C 180,E1 -17222.951,E2 -17222.951} C_VEL
LIN {X 0,Y 284.291,Z 270.572,A -85,B 0,C 180,E1 -17226.391,E2 -17226.391} C_VEL
LIN {X 0,Y 284.308,Z 270.571,A -85,B 0,C 180,E1 -17229.993,E2 -17229.993} C_VEL
LIN {X 0,Y 284.314,Z 270.568,A -85,B 0,C 180,E1 -17234.22,E2 -17234.22} C_VEL
LIN {X 0,Y 284.301,Z 270.57,A -85,B 0,C 180,E1 -17238.144,E2 -17238.144} C_VEL
LIN {X 0,Y 284.304,Z 270.569,A -85,B 0,C 180,E1 -17242.281,E2 -17242.281} C_VEL
LIN {X 0,Y 284.291,Z 270.575,A -85,B 0,C 180,E1 -17245.361,E2 -17245.361} C_VEL
LIN {X 0,Y 284.263,Z 270.575,A -85,B 0,C 180,E1 -17248.734,E2 -17248.734} C_VEL
LIN {X 0,Y 284.368,Z 270.563,A -85,B 0,C 180,E1 -17252.836,E2 -17252.836} C_VEL
LIN {X 0,Y 284.309,Z 270.569,A -85,B 0,C 180,E1 -17256.713,E2 -17256.713} C_VEL
LIN {X 0,Y 284.356,Z 270.559,A -85,B 0,C 180,E1 -17259.913,E2 -17259.913} C_VEL
LIN {X 0,Y 284.43,Z 270.555,A -85,B 0,C 180,E1 -17264.501,E2 -17264.501} C_VEL
LIN {X 0,Y 284.468,Z 270.552,A -85,B 0,C 180,E1 -17268.61,E2 -17268.61} C_VEL
LIN {X 0,Y 284.609,Z 270.53,A -85,B 0,C 180,E1 -17271.488,E2 -17271.488} C_VEL
LIN {X 0,Y 284.569,Z 270.538,A -85,B 0,C 180,E1 -17274.339,E2 -17274.339} C_VEL
LIN {X 0,Y 284.832,Z 270.494,A -85,B 0,C 180,E1 -17278.594,E2 -17278.594} C_VEL
LIN {X 0,Y 284.839,Z 270.5,A -85,B 0,C 180,E1 -17281.422,E2 -17281.422} C_VEL
LIN {X 0,Y 284.639,Z 270.527,A -85,B 0,C 180,E1 -17287.099,E2 -17287.099} C_VEL
LIN {X 0,Y 284.515,Z 270.547,A -85,B 0,C 180,E1 -17289.965,E2 -17289.965} C_VEL
LIN {X 0,Y 284.421,Z 270.556,A -85,B 0,C 180,E1 -17294.313,E2 -17294.313} C_VEL
LIN {X 0,Y 284.323,Z 270.567,A -85,B 0,C 180,E1 -17298.751,E2 -17298.751} C_VEL
LIN {X 0,Y 284.334,Z 270.567,A -85,B 0,C 180,E1 -17299.971,E2 -17299.971} C_VEL
LIN {X 0,Y 283.712,Z 270.651,A -85,B 0,C 180,E1 -17301.154,E2 -17301.154} C_VEL
LIN {X 0,Y 280.832,Z 271.011,A -85,B 0,C 180,E1 -17303.079,E2 -17303.079} C_VEL
LIN {X 0,Y 278.36,Z 271.314,A -85,B 0,C 180,E1 -17304.643,E2 -17304.643} C_VEL
LIN {X 0,Y 277.303,Z 271.443,A -85,B 0,C 180,E1 -17305.857,E2 -17305.857} C_VEL
LIN {X 0,Y 277.221,Z 271.451,A -85,B 0,C 180,E1 -17306.268,E2 -17306.268} C_VEL
LIN {X 0,Y 277.24,Z 271.453,A -85,B 0,C 180,E1 -17310.472,E2 -17310.472} C_VEL
LIN {X 0,Y 277.273,Z 271.712,A -85,B 0,C 180,E1 -17312.168,E2 -17312.168} C_VEL
LIN {X 0,Y 277.586,Z 273.785,A -85,B 0,C 180,E1 -17315.887,E2 -17315.887} C_VEL
LIN {X 0,Y 277.855,Z 275.834,A -85,B 0,C 180,E1 -17319.231,E2 -17319.231} C_VEL
LIN {X 0,Y 278.243,Z 278.386,A -85,B 0,C 180,E1 -17323.007,E2 -17323.007} C_VEL
LIN {X 0,Y 278.478,Z 280.596,A -85,B 0,C 180,E1 -17326.052,E2 -17326.052} C_VEL
LIN {X 0,Y 278.331,Z 283.135,A -85,B 0,C 180,E1 -17329.254,E2 -17329.254} C_VEL
LIN {X 0,Y 277.828,Z 286,A -85,B 0,C 180,E1 -17332.62,E2 -17332.62} C_VEL
LIN {X 0,Y 277.269,Z 289.118,A -85,B 0,C 180,E1 -17336.108,E2 -17336.108} C_VEL
LIN {X 0,Y 276.747,Z 292.493,A -85,B 0,C 180,E1 -17339.715,E2 -17339.715} C_VEL
LIN {X 0,Y 276.222,Z 296.1,A -85,B 0,C 180,E1 -17343.406,E2 -17343.406} C_VEL
LIN {X 0,Y 278.422,Z 304.278,A -85,B 0,C 180,E1 -17344.007,E2 -17344.007} C_VEL
LIN {X 0,Y 280.903,Z 314.602,A -85,B 0,C 180,E1 -17344.906,E2 -17344.906} C_VEL
LIN {X 0,Y 282.75,Z 324.343,A -85,B 0,C 180,E1 -17345.886,E2 -17345.886} C_VEL
LIN {X 0,Y 283.844,Z 333.518,A -85,B 0,C 180,E1 -17346.925,E2 -17346.925} C_VEL
LIN {X 0,Y 284.502,Z 342.495,A -85,B 0,C 180,E1 -17348.093,E2 -17348.093} C_VEL
LIN {X 0,Y 284.473,Z 346.338,A -85,B 0,C 180,E1 -17348.63,E2 -17348.63} C_VEL
LIN {X 0,Y 282.41,Z 357.837,A -85,B 0,C 180,E1 -17350.37,E2 -17350.37} C_VEL
LIN {X 0,Y 280.964,Z 365.95,A -85,B 0,C 180,E1 -17351.918,E2 -17351.918} C_VEL
LIN {X 0,Y 279.632,Z 373.186,A -85,B 0,C 180,E1 -17353.576,E2 -17353.576} C_VEL
LIN {X 0,Y 278.379,Z 379.726,A -85,B 0,C 180,E1 -17355.377,E2 -17355.377} C_VEL
LIN {X 0,Y 277.464,Z 384.228,A -85,B 0,C 180,E1 -17356.823,E2 -17356.823} C_VEL
LIN {X 0,Y 276.523,Z 389.726,A -85,B 0,C 180,E1 -17359.011,E2 -17359.011} C_VEL
LIN {X 0,Y 275.852,Z 394.055,A -85,B 0,C 180,E1 -17361.207,E2 -17361.207} C_VEL
LIN {X 0,Y 275.543,Z 396.425,A -85,B 0,C 180,E1 -17362.673,E2 -17362.673} C_VEL
LIN {X 0,Y 275.339,Z 398.773,A -85,B 0,C 180,E1 -17364.598,E2 -17364.598} C_VEL
LIN {X 0,Y 275.271,Z 400.681,A -85,B 0,C 180,E1 -17367.073,E2 -17367.073} C_VEL
LIN {X 0,Y 275.264,Z 401.272,A -85,B 0,C 180,E1 -17368.537,E2 -17368.537} C_VEL
LIN {X 0,Y 275.264,Z 401.272,A -85,B 0,C 180,E1 -17371.463,E2 -17371.463} C_VEL
LIN {X 0,Y 275.271,Z 400.681,A -85,B 0,C 180,E1 -17372.927,E2 -17372.927} C_VEL
LIN {X 0,Y 275.373,Z 398.228,A -85,B 0,C 180,E1 -17375.859,E2 -17375.859} C_VEL
LIN {X 0,Y 275.677,Z 395.273,A -85,B 0,C 180,E1 -17378.06,E2 -17378.06} C_VEL
LIN {X 0,Y 276.259,Z 391.281,A -85,B 0,C 180,E1 -17380.258,E2 -17380.258} C_VEL
LIN {X 0,Y 277.103,Z 386.146,A -85,B 0,C 180,E1 -17382.449,E2 -17382.449} C_VEL
LIN {X 0,Y 278.157,Z 380.882,A -85,B 0,C 180,E1 -17384.261,E2 -17384.261} C_VEL
LIN {X 0,Y 279.339,Z 374.562,A -85,B 0,C 180,E1 -17386.066,E2 -17386.066} C_VEL
LIN {X 0,Y 280.56,Z 368.611,A -85,B 0,C 180,E1 -17387.493,E2 -17387.493} C_VEL
LIN {X 0,Y 281.724,Z 361.678,A -85,B 0,C 180,E1 -17388.923,E2 -17388.923} C_VEL
LIN {X 0,Y 283.186,Z 353.496,A -85,B 0,C 180,E1 -17390.331,E2 -17390.331} C_VEL
LIN {X 0,Y 284.617,Z 344.984,A -85,B 0,C 180,E1 -17391.549,E2 -17391.549} C_VEL
LIN {X 0,Y 284.091,Z 336.237,A -85,B 0,C 180,E1 -17392.736,E2 -17392.736} C_VEL
LIN {X 0,Y 283.069,Z 326.562,A -85,B 0,C 180,E1 -17393.873,E2 -17393.873} C_VEL
LIN {X 0,Y 281.363,Z 316.756,A -85,B 0,C 180,E1 -17394.887,E2 -17394.887} C_VEL
LIN {X 0,Y 279.008,Z 306.549,A -85,B 0,C 180,E1 -17395.806,E2 -17395.806} C_VEL
LIN {X 0,Y 276.313,Z 296.873,A -85,B 0,C 180,E1 -17396.555,E2 -17396.555} C_VEL
LIN {X 0,Y 276.221,Z 296.002,A -85,B 0,C 180,E1 -17396.644,E2 -17396.644} C_VEL
LIN {X 0,Y 276.772,Z 292.249,A -85,B 0,C 180,E1 -17400.52,E2 -17400.52} C_VEL
LIN {X 0,Y 277.274,Z 289.116,A -85,B 0,C 180,E1 -17403.891,E2 -17403.891} C_VEL
LIN {X 0,Y 277.836,Z 285.967,A -85,B 0,C 180,E1 -17407.379,E2 -17407.379} C_VEL
LIN {X 0,Y 278.353,Z 282.892,A -85,B 0,C 180,E1 -17411.03,E2 -17411.03} C_VEL
LIN {X 0,Y 278.484,Z 280.579,A -85,B 0,C 180,E1 -17413.947,E2 -17413.947} C_VEL
LIN {X 0,Y 278.235,Z 278.284,A -85,B 0,C 180,E1 -17417.097,E2 -17417.097} C_VEL
LIN {X 0,Y 277.856,Z 275.83,A -85,B 0,C 180,E1 -17420.769,E2 -17420.769} C_VEL
LIN {X 0,Y 277.558,Z 273.611,A -85,B 0,C 180,E1 -17424.374,E2 -17424.374} C_VEL
LIN {X 0,Y 277.273,Z 271.712,A -85,B 0,C 180,E1 -17427.832,E2 -17427.832} C_VEL
LIN {X 0,Y 277.226,Z 271.454,A -85,B 0,C 180,E1 -17431.198,E2 -17431.198} C_VEL
LIN {X 0,Y 277.24,Z 271.456,A -85,B 0,C 180,E1 -17434.465,E2 -17434.465} C_VEL
LIN {X 0,Y 277.255,Z 271.451,A -85,B 0,C 180,E1 -17437.645,E2 -17437.645} C_VEL
LIN {X 0,Y 277.283,Z 271.446,A -85,B 0,C 180,E1 -17440.754,E2 -17440.754} C_VEL
LIN {X 0,Y 277.375,Z 271.432,A -85,B 0,C 180,E1 -17445.315,E2 -17445.315} C_VEL
LIN {X 0,Y 277.455,Z 271.425,A -85,B 0,C 180,E1 -17449.779,E2 -17449.779} C_VEL
LIN {X 0,Y 277.598,Z 271.404,A -85,B 0,C 180,E1 -17452.72,E2 -17452.72} C_VEL
LIN {X 0,Y 277.805,Z 271.376,A -85,B 0,C 180,E1 -17458.542,E2 -17458.542} C_VEL
LIN {X 0,Y 277.799,Z 271.368,A -85,B 0,C 180,E1 -17461.441,E2 -17461.441} C_VEL
LIN {X 0,Y 277.604,Z 271.406,A -85,B 0,C 180,E1 -17467.263,E2 -17467.263} C_VEL
LIN {X 0,Y 277.444,Z 271.421,A -85,B 0,C 180,E1 -17470.204,E2 -17470.204} C_VEL
LIN {X 0,Y 277.393,Z 271.428,A -85,B 0,C 180,E1 -17474.667,E2 -17474.667} C_VEL
LIN {X 0,Y 277.297,Z 271.441,A -85,B 0,C 180,E1 -17479.227,E2 -17479.227} C_VEL
LIN {X 0,Y 277.272,Z 271.443,A -85,B 0,C 180,E1 -17483.915,E2 -17483.915} C_VEL
LIN {X 0,Y 277.296,Z 271.443,A -85,B 0,C 180,E1 -17487.495,E2 -17487.495} C_VEL
LIN {X 0,Y 277.244,Z 271.451,A -85,B 0,C 180,E1 -17490.473,E2 -17490.473} C_VEL
LIN {X 0,Y 277.222,Z 271.451,A -85,B 0,C 180,E1 -17493.887,E2 -17493.887} C_VEL
LIN {X 0,Y 277.25,Z 271.448,A -85,B 0,C 180,E1 -17497.459,E2 -17497.459} C_VEL
LIN {X 0,Y 277.228,Z 271.451,A -85,B 0,C 180,E1 -17501.219,E2 -17501.219} C_VEL
LIN {X 0,Y 277.247,Z 271.448,A -85,B 0,C 180,E1 -17505.201,E2 -17505.201} C_VEL
LIN {X 0,Y 277.252,Z 271.447,A -85,B 0,C 180,E1 -17509.488,E2 -17509.488} C_VEL
LIN {X 0,Y 277.232,Z 271.452,A -85,B 0,C 180,E1 -17512.526,E2 -17512.526} C_VEL
LIN {X 0,Y 277.2,Z 271.458,A -85,B 0,C 180,E1 -17516.098,E2 -17516.098} C_VEL
LIN {X 0,Y 277.213,Z 271.455,A -85,B 0,C 180,E1 -17519.533,E2 -17519.533} C_VEL
LIN {X 0,Y 277.286,Z 271.446,A -85,B 0,C 180,E1 -17523.182,E2 -17523.182} C_VEL
LIN {X 0,Y 278.384,Z 274.45,A -85,B 0,C 180,E1 -17523.384,E2 -17523.384} C_VEL
LIN {X 0,Y 284.761,Z 287.942,A -85,B 0,C 180,E1 -17524.548,E2 -17524.548} C_VEL
LIN {X 0,Y 289.378,Z 296.305,A -85,B 0,C 180,E1 -17525.478,E2 -17525.478} C_VEL
LIN {X 0,Y 295.816,Z 305.978,A -85,B 0,C 180,E1 -17526.777,E2 -17526.777} C_VEL
LIN {X 0,Y 303.971,Z 316.256,A -85,B 0,C 180,E1 -17528.408,E2 -17528.408} C_VEL
LIN {X 0,Y 312.16,Z 325.71,A -85,B 0,C 180,E1 -17530.096,E2 -17530.096} C_VEL
LIN {X 0,Y 319.476,Z 333.585,A -85,B 0,C 180,E1 -17531.777,E2 -17531.777} C_VEL
LIN {X 0,Y 325.523,Z 339.724,A -85,B 0,C 180,E1 -17533.289,E2 -17533.289} C_VEL
LIN {X 0,Y 331.392,Z 345.391,A -85,B 0,C 180,E1 -17534.943,E2 -17534.943} C_VEL
LIN {X 0,Y 335.933,Z 349.464,A -85,B 0,C 180,E1 -17536.348,E2 -17536.348} C_VEL
LIN {X 0,Y 340.85,Z 354.085,A -85,B 0,C 180,E1 -17538.101,E2 -17538.101} C_VEL
LIN {X 0,Y 344.309,Z 356.797,A -85,B 0,C 180,E1 -17539.414,E2 -17539.414} C_VEL
LIN {X 0,Y 347.118,Z 359.064,A -85,B 0,C 180,E1 -17540.679,E2 -17540.679} C_VEL
LIN {X 0,Y 349.214,Z 361.202,A -85,B 0,C 180,E1 -17541.902,E2 -17541.902} C_VEL
LIN {X 0,Y 351.11,Z 362.92,A -85,B 0,C 180,E1 -17543.102,E2 -17543.102} C_VEL
LIN {X 0,Y 353.018,Z 364.286,A -85,B 0,C 180,E1 -17544.407,E2 -17544.407} C_VEL
LIN {X 0,Y 354.421,Z 365.08,A -85,B 0,C 180,E1 -17545.451,E2 -17545.451} C_VEL
LIN {X 0,Y 355.78,Z 365.643,A -85,B 0,C 180,E1 -17546.603,E2 -17546.603} C_VEL
LIN {X 0,Y 356.801,Z 365.967,A -85,B 0,C 180,E1 -17547.742,E2 -17547.742} C_VEL
LIN {X 0,Y 357.494,Z 366.079,A -85,B 0,C 180,E1 -17548.874,E2 -17548.874} C_VEL
LIN {X 0,Y 357.742,Z 366.095,A -85,B 0,C 180,E1 -17550,E2 -17550} C_VEL
LIN {X 0,Y 357.49,Z 366.068,A -85,B 0,C 180,E1 -17551.126,E2 -17551.126} C_VEL
LIN {X 0,Y 356.798,Z 365.952,A -85,B 0,C 180,E1 -17552.258,E2 -17552.258} C_VEL
LIN {X 0,Y 355.774,Z 365.635,A -85,B 0,C 180,E1 -17553.397,E2 -17553.397} C_VEL
LIN {X 0,Y 354.418,Z 365.091,A -85,B 0,C 180,E1 -17554.549,E2 -17554.549} C_VEL
LIN {X 0,Y 352.868,Z 364.198,A -85,B 0,C 180,E1 -17555.715,E2 -17555.715} C_VEL
LIN {X 0,Y 351.097,Z 362.91,A -85,B 0,C 180,E1 -17556.898,E2 -17556.898} C_VEL
